(* CODESYS project system_dk.library
   Company: Beckhoff - DK
   DefaultNamespace: Tc3_System_DK
   Title: Tc3_System_DK
   Placeholder: Tc3_System_DK
   Author: HCP
   Version: 3.3.2.4

Project tree, tasks and I/O mapping:
  libraries: Tc2_EtherCAT, * (Beckhoff Automation GmbH); Tc2_IoFunctions, * (Beckhoff Automation GmbH); Tc2_Standard, * (Beckhoff Automation GmbH); Tc2_SUPS, * (Beckhoff Automation GmbH); Tc2_System, * (Beckhoff Automation GmbH); Tc2_Utilities, * (Beckhoff Automation GmbH); Tc3_Interfaces, * (Beckhoff Automation GmbH); Tc3_Module, * (Beckhoff Automation GmbH)
  DUTs/
  GVLs/
  POUs/
    BASE/
      FBs/
        [obsolete]/
          Basic/
            DUTs/
              data type ST_Basic
              data type ST_Basic_Status
            ITFs/
              interface I_Basic: M_nError, M_nReset, P_bAuto, P_bError, P_bManual, P_bReady, P_bReset, P_nErrorID
            function block FB_Basic [ST]: M_nError, M_nReset, P_bAuto, P_bError, P_bManual, P_bReady, P_bReset, P_nErrorID
        Base/
          DUTs/
            data type ST_Base
            data type ST_Base_Status
          ITFs/
            interface I_Base: M_nError, M_nReset, P_bError, P_bReady, P_bReset, P_nErrorID
          function block FB_Base [ST]: M_nError, M_nReset, P_bError, P_bReady, P_bReset, P_nErrorID
      GVLs/
        global variables GVL_Base
    SYSTEM/
      FBs/
        EtherCAT/
          DUTs/
            HW/
              data type ST_EtherCAT_HW_IN
              data type ST_EtherCAT_HW_TerminalDiagInfo
            data type ST_EtherCAT_DiagDk
            data type ST_EtherCAT_HW_Diag
          GVLs/
            global variables GVL_EtherCAT_Diag
          ITFs/
            interface I_EtherCAT_DiagDk: M_nCyclic, P_bEtherCAT_Ok, P_bWcError, P_nCfgSlaveCount, P_nDevState, P_nSlaveCounts
          function block FB_EtherCAT_DiagDk [ST]: M_nCyclic, M_sGetToken, P_bEtherCAT_Ok, P_bWcError, P_nCfgSlaveCount, P_nDevState, P_nSlaveCounts
        NovRam/
          DUTs/
            data type ST_NovRamDK
          ITFs/
            interface I_NovRamDK: M_nEnable
          function block FB_NovRamDK [ST]: M_nEnable, M_nRead, M_nWrite
        Persistent/
          DUTs/
            data type ST_WritePersistentDataDK
          ITFs/
            interface I_WritePersistentDataDK: M_n1_Second_UPS, M_nEnable, M_nWrite, P_bBusy, P_bPowerFailDetect, P_ePersistentMode, P_eSUPS_Mode, P_nWriteCNT
          function block FB_WritePersistentDataDK [ST]: M_n1_Second_UPS, M_nEnable, M_nWrite, P_bBusy, P_bPowerFailDetect, P_ePersistentMode, P_eSUPS_Mode, P_nWriteCNT
        System/
          DUTs/
            data type ST_SystemDK
          ITFs/
            interface I_SystemDK: M_nCerHost, M_nEnable, M_nGetTimeStampInMs, P_bIs_ARM, P_bIs_CE_Device, P_bIs_x64, P_bIs_x86, P_nAdsPort, P_nCycleTime, P_sHardwareSerialNumber, P_stDeviceIdentificationEx, P_sTwinCAT_Version
          function block FB_SystemDK [ST]: M_nCerHost, M_nEnable, M_nGetTimeStampInMs, P_bIs_ARM, P_bIs_CE_Device, P_bIs_x64, P_bIs_x86, P_nAdsPort, P_nCycleTime, P_sHardwareSerialNumber, P_stDeviceIdentificationEx, P_sTwinCAT_Version
  Version/
    global variables Global_Version
  VISUs/
*)

// POUs/BASE/FBs/[obsolete]/Basic/DUTs/ST_Basic
TYPE ST_Basic :
STRUCT
	bAuto: BOOL;
	bManual: BOOL;
	bReady: BOOL;
	bReset: BOOL;
	bError: BOOL;
	nErrorID: UDINT;
	nStatus: UDINT;	
	arr_nStatus: ARRAY[1..20] OF UDINT;
END_STRUCT
END_TYPE

// POUs/BASE/FBs/[obsolete]/Basic/DUTs/ST_Basic_Status
TYPE ST_Basic_Status :
STRUCT
	nError: UDINT;
	nReset:UDINT;
END_STRUCT
END_TYPE

// POUs/BASE/FBs/Base/DUTs/ST_Base
TYPE ST_Base :
STRUCT
	bReset: BOOL;
	bReady: BOOL;
	bError: BOOL;
	nErrorID: UDINT;
	arr_nStatus: ARRAY[1..20] OF UDINT;
END_STRUCT
END_TYPE

// POUs/BASE/FBs/Base/DUTs/ST_Base_Status
TYPE ST_Base_Status :
STRUCT
	nError: UDINT;
	nReset:UDINT;
END_STRUCT
END_TYPE

// POUs/SYSTEM/FBs/EtherCAT/DUTs/HW/ST_EtherCAT_HW_IN
TYPE ST_EtherCAT_HW_IN :
STRUCT
	AI_AmsNetId: AMSNETID;
	AI_nDevState: UINT;
	AI_nCfgSlaveCount: UINT;							
	AI_nSlaveCounts: UINT;								
	AI_nFrmXWcState: ARRAY[0..(GVL_EtherCAT_Diag.cMAX_NUMBERS_OF_EC_FRAMES -1)] OF UINT;
END_STRUCT
END_TYPE

// POUs/SYSTEM/FBs/EtherCAT/DUTs/HW/ST_EtherCAT_HW_TerminalDiagInfo
TYPE ST_EtherCAT_HW_TerminalDiagInfo :
STRUCT
	nAddr: UINT;
	sType: STRING(50);
	sName: STRING(50);
	nDeviceState: BYTE;
	nLinkState: BYTE;
	stTopologyDataEx: Tc2_EtherCAT.ST_TopologyDataEx;
END_STRUCT
END_TYPE

// POUs/SYSTEM/FBs/EtherCAT/DUTs/ST_EtherCAT_DiagDk
TYPE ST_EtherCAT_DiagDk EXTENDS ST_Basic:
STRUCT
	bEtherCAT_Ok: BOOL;				// ErtherCAT Ok signal
	bWcError: BOOL;
	nDevState: UINT;
	nCfgSlaveCount: UINT;							
	nSlaveCounts: UINT;								
END_STRUCT
END_TYPE

// POUs/SYSTEM/FBs/EtherCAT/DUTs/ST_EtherCAT_HW_Diag
TYPE ST_EtherCAT_HW_Diag :
STRUCT
	stAmsNetId: AMSNETID;			// EtherCAT Ams net id
	nState: WORD;					// EtherCAT master state
	sState: STRING;					// EtherCAT master state (string)
	nDevState: UINT;				// EtherCAT master DevState
	sDevState: STRING;				// EtherCAT master DevState (string)
	nCfgSlaveCount: UINT;			// Project configured slaves
	nSlaveCounts: UINT;				// Actual slave counts
	nMaxNumberOfSlaves: UINT;		// Max numbers of EtherCAT slaves
	bWcError: BOOL;					// Wc error
	bEtherCAT_Ok: BOOL;				// ErtherCAT Ok signal
	bReady: BOOL;					// Ready
	bError: BOOL;					// Error
	nErrorID: UDINT;				// Error ID
	arrFrmXWcState: ARRAY[0..(GVL_EtherCAT_Diag.cMAX_NUMBERS_OF_EC_FRAMES - 1)] OF UINT;		// EtherCAT master Wc state
	arrEcTerminalDiagInfo: ARRAY[1..GVL_EtherCAT_Diag.cMAX_NUMBERS_OF_EC_SLAVES] OF ST_EtherCAT_HW_TerminalDiagInfo;
END_STRUCT
END_TYPE

// POUs/SYSTEM/FBs/NovRam/DUTs/ST_NovRamDK
TYPE ST_NovRamDK EXTENDS ST_Basic :
STRUCT
	bEnable: BOOL;
END_STRUCT
END_TYPE

// POUs/SYSTEM/FBs/Persistent/DUTs/ST_WritePersistentDataDK
TYPE ST_WritePersistentDataDK EXTENDS ST_Basic :
STRUCT
	bWrite: BOOL;
	bBusy: BOOL;
	bPowerFailDetect: BOOL;
	nWriteCNT: UDINT;
END_STRUCT
END_TYPE

// POUs/SYSTEM/FBs/System/DUTs/ST_SystemDK
TYPE ST_SystemDK EXTENDS ST_Basic :
STRUCT
	bIs_CE_Device: BOOL;				// Is a CE Device
	bIs_ARM: BOOL;						// Is ARM runtime
	bIs_x86: BOOL;						// Is x86 runtime
	bIs_x64: BOOL;						// Is x64 runtime
	nAdsPort: UINT;						// Plc port nr
	nCycleTime: UDINT;					// Plc cycle time in 100nS
	bCerHost_Enable: BOOL;				// Enable CerHost
	bCerHost_Disable: BOOL;				// Disable CerHost
	sTwinCAT_Version: STRING(20);		// Runtime version
	sHardwareSerialNumber: STRING(20);	// Runtime hardware serial number
	stDeviceIdentificationEx: Tc2_Utilities.ST_DeviceIdentificationEx;		// Runtime info
END_STRUCT
END_TYPE

// POUs/BASE/GVLs/GVL_Base
VAR_GLOBAL CONSTANT
	cIDLE: UDINT:= 0;						//	0 = idle
	cCOUPLED: UDINT:= 1;					//	1 = coupled
	cSTARTING: UDINT:= 2;					//	2 = starting
	cRUNNING: UDINT:= 3;					//	3 = running
	cABORTED: UDINT:= 4;					//	4 = aborted
	cNO_HARDWARE_CONNECTED: UDINT:= 5;		// 	5 = no hardware connected

	cPOINTER_OR_INDEX_ERROR: UDINT:= 7;		//	7 = pointer or index error
	cMAPPING_ERROR: UDINT:= 8;				//	8 = mapping error
	cPARAMETER_ERROR: UDINT:= 9;			//	9 = parameter error
	cCOMPLETE: UDINT:= 10;					//	10 = complete
END_VAR

// POUs/SYSTEM/FBs/EtherCAT/GVLs/GVL_EtherCAT_Diag
{attribute 'qualified_only'}
VAR_GLOBAL CONSTANT
	cMAX_NUMBERS_OF_EC_SLAVES: UINT:= 1000;		// Max numbers of EtherCAT slaves
	cMAX_NUMBERS_OF_EC_FRAMES: UINT:= 10;		// Max numbers of EtherCAT frames
END_VAR

// Version/Global_Version
{attribute 'TcGenerated'}
{attribute 'no-analysis'}
{attribute 'linkalways'}
// This function has been automatically generated from the project information.
VAR_GLOBAL CONSTANT
	{attribute 'const_non_replaced'}
	stLibVersion_Tc3_System_DK : ST_LibVersion := (iMajor := 3, iMinor := 3, iBuild := 2, iRevision := 4, sVersion := '3.3.2.4');
END_VAR

// POUs/BASE/FBs/[obsolete]/Basic/ITFs/I_Basic
INTERFACE I_Basic

//	The result of the method is an unsigned double integer
//	0 = idle 
//	1 = coupled
//	2 = starting
//	3 = running
//	4 = aborted
// 	5 = no hardware connected
//  6 = Spare
//	7 = pointer or index error
//	8 = mapping error
//	9 = parameter error
//	10 = complete
//	Any other number = ErrorID
METHOD PUBLIC M_nError : UDINT
VAR_INPUT
	nErrorID: UDINT;
END_VAR
END_METHOD

//	The result of the method is an unsigned double integer
//	0 = idle 
//	1 = coupled
//	2 = starting
//	3 = running
//	4 = aborted
// 	5 = no hardware connected
//  6 = Spare
//	7 = pointer or index error
//	8 = mapping error
//	9 = parameter error
//	10 = complete
//	Any other number = ErrorID
METHOD PUBLIC M_nReset : UDINT
VAR_INPUT
	bExecute: BOOL;
END_VAR
END_METHOD

PROPERTY PUBLIC P_bAuto : BOOL
GET
END_GET
SET
END_SET
END_PROPERTY

PROPERTY PUBLIC P_bError : BOOL
GET
END_GET
END_PROPERTY

PROPERTY PUBLIC P_bManual : BOOL
GET
END_GET
SET
END_SET
END_PROPERTY

PROPERTY PUBLIC P_bReady : BOOL
GET
END_GET
SET
END_SET
END_PROPERTY

PROPERTY PUBLIC P_bReset : BOOL
GET
END_GET
END_PROPERTY

PROPERTY PUBLIC P_nErrorID : UDINT
GET
END_GET
END_PROPERTY

END_INTERFACE

// POUs/BASE/FBs/[obsolete]/Basic/FB_Basic
//------------------------------------------------------------------------------------------
//                                                                                        	
//***************************** Beckhoff TwinCAT Examples **********************************
//                                                                                        	
//************************************* WARNING ********************************************
// This program is only an example. If it is used as a control program in any real        	
// application, Beckhoff is not responsible for any malfunction, loss or damage           	
// which could arise by using this program!                                               	
//                                                                                        	
//*************************************  Program Info. *************************************
//                                                                                        	
// PLC program name:       	FB_Basic (FB)               	                           	
// Hardware platform:      	TwinCat v3.1.4012				                          	
// Modified by:            	Hans Chr. Pallesen 			                                  	
// Email:					h.pallesen@beckhoff.com	                                  	
//                                                                                        	
// ======================================================================================== 
//         Version       Date                        Remarks                              	
// ======================================================================================== 
//         1.0           17 feb 2013                 First release of this example        	
//         1.1           05 aug 2013                 Next release of this example        	
//         1.2           10 dec 2013                 Next release of this example        	
//         1.3           12 mar 2014                 Next release of this example        	
//         1.4           28 mar 2014                 Next release of this example        	
//         1.5           02 jun 2014                 Next release of this example        	
// ======================================================================================== 
//                                                                                        	
//******************************* Aims OF this PLC PROGRAM *********************************
//                                                                                        	
// Basic FB  						 			                               	
//																	                      	
//                                                                                        	
//----------------------------------------------------------------------------------------- 
FUNCTION_BLOCK FB_Basic IMPLEMENTS I_Basic
VAR
	_iIdx: INT;		// Temporary variabel - Index pointer
	
//*************************
// Property variables
//*************************
	_bReset: BOOL;
	_bAuto: BOOL := TRUE;
	_bManual: BOOL;
	_bError: BOOL;
	_nErrorID: UDINT;
	_bReady: BOOL;
	
//*************************
// Methods variable
//*************************
	_nResetState: UINT;
END_VAR

//	The result of the method is an unsigned double integer
//	0 = idle 
//	1 = coupled
//	2 = starting
//	3 = running
//	4 = aborted
// 	5 = no hardware connected
//  6 = Spare
//	7 = pointer or index error
//	8 = mapping error
//	9 = parameter error
//	10 = complete
//	Any other number = ErrorID
METHOD PUBLIC M_nError : UDINT
VAR_INPUT
	nErrorID: UDINT;
END_VAR
//**********************************
// Update error
//**********************************
IF _nResetState = 0 OR _nResetState = 4 THEN
	IF NOT _bError THEN
		_nErrorID:= nErrorID;
		_bError:= TRUE;
	END_IF
END_IF

M_nError:= cCOMPLETE;
END_METHOD

//	The result of the method is an unsigned double integer
//	0 = idle 
//	1 = coupled
//	2 = starting
//	3 = running
//	4 = aborted
// 	5 = no hardware connected
//  6 = Spare
//	7 = pointer or index error
//	8 = mapping error
//	9 = parameter error
//	10 = complete
//	Any other number = ErrorID
METHOD PUBLIC M_nReset : UDINT
VAR_INPUT
	bExecute: BOOL;
END_VAR
// Reset handling
CASE _nResetState OF

	000:	// Wait for execute
			M_nReset:= cIDLE;
			IF bExecute THEN
				_bReset:= TRUE;
				_nResetState:= _nResetState +1;
			ELSE
				_bReset:= FALSE;
			END_IF

	001:	// Reset update
			M_nReset:= cRUNNING;
			_nResetState:= _nResetState +1;
		
	002:	// Reset error flag
			M_nReset:= cRUNNING;
			_bError:= FALSE;
			_nErrorID:= 16#00;
			_nResetState:= _nResetState +1;
	
	003:	// Reset update
			M_nReset:= cRUNNING;
			_nResetState:= _nResetState +1;
		
	004:	// Wait for not execute
			IF bExecute THEN
				M_nReset:= cCOMPLETE;
			ELSE
				M_nReset:= cCOMPLETE;
				_bReset:= FALSE;
				_nResetState:= 000;
			END_IF

ELSE
		_nResetState:= 000;
END_CASE
END_METHOD

PROPERTY PUBLIC P_bAuto : BOOL
GET
P_bAuto:= _bAuto;
END_GET
SET
_bAuto:= P_bAuto;
END_SET
END_PROPERTY

PROPERTY PUBLIC P_bError : BOOL
GET
P_bError:= _bError;
END_GET
END_PROPERTY

PROPERTY PUBLIC P_bManual : BOOL
GET
P_bManual:= _bManual;
END_GET
SET
_bManual:= P_bManual;
END_SET
END_PROPERTY

PROPERTY PUBLIC P_bReady : BOOL
GET
P_bReady:= _bReady;
END_GET
SET
PUBLIC 
VAR
END_VAR
_bReady:= P_bReady;
END_SET
END_PROPERTY

PROPERTY PUBLIC P_bReset : BOOL
GET
P_bReset:= _bReset;
END_GET
END_PROPERTY

PROPERTY PUBLIC P_nErrorID : UDINT
GET
P_nErrorID:= _nErrorID;
END_GET
END_PROPERTY

END_FUNCTION_BLOCK

// POUs/BASE/FBs/Base/ITFs/I_Base
INTERFACE I_Base

//	The result of the method is an unsigned double integer
//	0 = idle 
//	1 = coupled
//	2 = starting
//	3 = running
//	4 = aborted
// 	5 = no hardware connected
//  6 = Spare
//	7 = pointer or index error
//	8 = mapping error
//	9 = parameter error
//	10 = complete
//	Any other number = ErrorID
METHOD PUBLIC M_nError : UDINT
VAR_INPUT
	nErrorID: UDINT;
END_VAR
END_METHOD

//	The result of the method is an unsigned double integer
//	0 = idle 
//	1 = coupled
//	2 = starting
//	3 = running
//	4 = aborted
// 	5 = no hardware connected
//  6 = Spare
//	7 = pointer or index error
//	8 = mapping error
//	9 = parameter error
//	10 = complete
//	Any other number = ErrorID
METHOD PUBLIC M_nReset : UDINT
VAR_INPUT
	bExecute: BOOL;
END_VAR
END_METHOD

PROPERTY PUBLIC P_bError : BOOL
GET
END_GET
END_PROPERTY

PROPERTY PUBLIC P_bReady : BOOL
GET
END_GET
SET
END_SET
END_PROPERTY

PROPERTY PUBLIC P_bReset : BOOL
GET
END_GET
END_PROPERTY

PROPERTY PUBLIC P_nErrorID : UDINT
GET
END_GET
END_PROPERTY

END_INTERFACE

// POUs/BASE/FBs/Base/FB_Base
//------------------------------------------------------------------------------------------
//                                                                                        	
//***************************** Beckhoff TwinCAT Examples **********************************
//                                                                                        	
//************************************* WARNING ********************************************
// This program is only an example. If it is used as a control program in any real        	
// application, Beckhoff is not responsible for any malfunction, loss or damage           	
// which could arise by using this program!                                               	
//                                                                                        	
//*************************************  Program Info. *************************************
//                                                                                        	
// PLC program name:       	FB_Basic (FB)               	                           	
// Hardware platform:      	TwinCat v3.1.4020				                          	
// Modified by:            	Hans Chr. Pallesen 			                                  	
// Email:					h.pallesen@beckhoff.com	                                  	
//                                                                                        	
// ======================================================================================== 
//         Version       Date                        Remarks                              	
// ======================================================================================== 
//         1.0           02 mar 2019                 First release of this example        	
// ======================================================================================== 
//                                                                                        	
//******************************* Aims OF this PLC PROGRAM *********************************
//                                                                                        	
// Base FB  						 			                               	
//																	                      	
//                                                                                        	
//----------------------------------------------------------------------------------------- 
FUNCTION_BLOCK FB_Base IMPLEMENTS I_Base
VAR
	
//*************************
// Property variables
//*************************
	_bReset: BOOL;
	_bError: BOOL;
	_nErrorID: UDINT;
	_bReady: BOOL;

//*************************
// Methodes variables
//*************************
	_nResetState: UINT;
	
END_VAR

//	The result of the method is an unsigned double integer
//	0 = idle 
//	1 = coupled
//	2 = starting
//	3 = running
//	4 = aborted
// 	5 = no hardware connected
//  6 = Spare
//	7 = pointer or index error
//	8 = mapping error
//	9 = parameter error
//	10 = complete
//	Any other number = ErrorID
METHOD PUBLIC M_nError : UDINT
VAR_INPUT
	nErrorID: UDINT;
END_VAR
//**********************************
// Update error
//**********************************
IF _nResetState = 0 OR _nResetState = 4 THEN
	IF NOT _bError THEN
		_nErrorID:= nErrorID;
		_bError:= TRUE;
	END_IF
END_IF

M_nError:= cCOMPLETE;
END_METHOD

//	The result of the method is an unsigned double integer
//	0 = idle 
//	1 = coupled
//	2 = starting
//	3 = running
//	4 = aborted
// 	5 = no hardware connected
//  6 = Spare
//	7 = pointer or index error
//	8 = mapping error
//	9 = parameter error
//	10 = complete
//	Any other number = ErrorID
METHOD PUBLIC M_nReset : UDINT
VAR_INPUT
	bExecute: BOOL;
END_VAR
VAR_INST
	_FB_Base_M_nReset_nState: UINT;
END_VAR
// Reset handling
CASE _FB_Base_M_nReset_nState OF

	000:	// Wait for execute
			M_nReset:= cIDLE;
			IF bExecute THEN
				_bReset:= TRUE;
				_FB_Base_M_nReset_nState:= _FB_Base_M_nReset_nState +1;
			ELSE
				_bReset:= FALSE;
			END_IF

	001:	// Reset update
			M_nReset:= cRUNNING;
			_FB_Base_M_nReset_nState:= _FB_Base_M_nReset_nState +1;
		
	002:	// Reset error flag
			M_nReset:= cRUNNING;
			_bError:= FALSE;
			_nErrorID:= 16#00;
			_FB_Base_M_nReset_nState:= _FB_Base_M_nReset_nState +1;
	
	003:	// Reset update
			M_nReset:= cRUNNING;
			_FB_Base_M_nReset_nState:= _FB_Base_M_nReset_nState +1;
		
	004:	// Wait for not execute
			IF bExecute THEN
				M_nReset:= cCOMPLETE;
			ELSE
				M_nReset:= cCOMPLETE;
				_bReset:= FALSE;
				_FB_Base_M_nReset_nState:= 000;
			END_IF

ELSE
		_FB_Base_M_nReset_nState:= 000;
END_CASE
END_METHOD

{attribute 'monitoring' := 'variable'}
PROPERTY PUBLIC P_bError : BOOL
GET
P_bError:= _bError;
END_GET
END_PROPERTY

{attribute 'monitoring' := 'variable'}
PROPERTY PUBLIC P_bReady : BOOL
GET
P_bReady:= _bReady;
END_GET
SET
PUBLIC 
VAR
END_VAR
_bReady:= P_bReady;
END_SET
END_PROPERTY

{attribute 'monitoring' := 'variable'}
PROPERTY PUBLIC P_bReset : BOOL
GET
P_bReset:= _bReset;
END_GET
END_PROPERTY

{attribute 'monitoring' := 'variable'}
PROPERTY PUBLIC P_nErrorID : UDINT
GET
P_nErrorID:= _nErrorID;
END_GET
END_PROPERTY

END_FUNCTION_BLOCK

// POUs/SYSTEM/FBs/EtherCAT/ITFs/I_EtherCAT_DiagDk
INTERFACE I_EtherCAT_DiagDk EXTENDS I_Basic

//	The result of the method is an unsigned double integer
//	0 = idle 
//	1 = coupled
//	2 = starting
//	3 = running
//	4 = aborted
// 	5 = no hardware connected
//  6 = Spare
//	7 = pointer or index error
//	8 = mapping error
//	9 = parameter error
//	10 = complete
//	Any other number = ErrorID
METHOD PUBLIC M_nCyclic : UDINT
VAR_INPUT
	bEnable: BOOL;
	pEtherCAT_Diag: POINTER TO ST_EtherCAT_HW_Diag;	
END_VAR
END_METHOD

PROPERTY PUBLIC P_bEtherCAT_Ok : BOOL
GET
END_GET
SET
END_SET
END_PROPERTY

PROPERTY PUBLIC P_bWcError : bool
GET
END_GET
END_PROPERTY

PROPERTY PUBLIC P_nCfgSlaveCount : UINT
GET
END_GET
END_PROPERTY

PROPERTY PUBLIC P_nDevState : UINT
GET
END_GET
END_PROPERTY

PROPERTY PUBLIC P_nSlaveCounts : UINT
GET
END_GET
END_PROPERTY

END_INTERFACE

// POUs/SYSTEM/FBs/EtherCAT/FB_EtherCAT_DiagDk
//------------------------------------------------------------------------------------------
//                                                                                        	
//***************************** Beckhoff TwinCAT Examples **********************************
//                                                                                        	
//************************************* WARNING ********************************************
// This program is only an example. If it is used as a control program in any real        	
// application, Beckhoff is not responsible for any malfunction, loss or damage           	
// which could arise by using this program!                                               	
//                                                                                        	
//*************************************  Program Info. *************************************
//                                                                                        	
// PLC program name:       	FB_EtherCAT_Diag (FB)                                          	
// Hardware platform:      	TwinCAT v3.1.4022				                          	
// Modified by:            	Hans Chr. Pallesen 			                                  	
// Email:					h.pallesen@beckhoff.com	                                  	
//                                                                                        	
// ======================================================================================== 
//         Version       Date                        Remarks                              	
// ======================================================================================== 
//         1.0           12 dec 2016                 First release of this example        	
// ======================================================================================== 
//                                                                                        	
//******************************* Aims OF this PLC PROGRAM *********************************
//                                                                                        	
// EtherCAT diagnose				 			                                      	
//																	                      	
//                                                                                        	
//----------------------------------------------------------------------------------------- 
FUNCTION_BLOCK FB_EtherCAT_DiagDk EXTENDS FB_Basic IMPLEMENTS I_EtherCAT_DiagDk
VAR
	bFirstScan: BOOL:= TRUE;
	stIN AT %I*: ST_EtherCAT_HW_IN;
	
	_pEtherCAT_Diag: POINTER TO ST_EtherCAT_HW_Diag;	
	_bWcError: BOOL;
	_nDeviceNumber: UINT:= 1;
	_nSlaves: UINT;
	
	arrEcSlaveConfigData: ARRAY[1..GVL_EtherCAT_Diag.cMAX_NUMBERS_OF_EC_SLAVES] OF Tc2_EtherCAT.ST_EcSlaveConfigData;
	arrEcSlaveState: ARRAY[1..GVL_EtherCAT_Diag.cMAX_NUMBERS_OF_EC_SLAVES] OF Tc2_EtherCAT.ST_EcSlaveState;
	arrTopologyDataEx: ARRAY[1..GVL_EtherCAT_Diag.cMAX_NUMBERS_OF_EC_SLAVES] OF Tc2_EtherCAT.ST_TopologyDataEx;
	arrEcSlaveName: ARRAY[1..GVL_EtherCAT_Diag.cMAX_NUMBERS_OF_EC_SLAVES] OF STRING;;
	arrFrmXWcStateOld: ARRAY[0..(GVL_EtherCAT_Diag.cMAX_NUMBERS_OF_EC_FRAMES -1)] OF UINT;
	arrFrmXWcStateInit: ARRAY[0..(GVL_EtherCAT_Diag.cMAX_NUMBERS_OF_EC_FRAMES -1)] OF UINT;
	
	fbEcGetMasterState: Tc2_EtherCAT.FB_EcGetMasterState;
	fbEcGetConfSlaves: Tc2_EtherCAT.FB_EcGetConfSlaves;
	fbEcGetAllSlaveStates: Tc2_EtherCAT.FB_EcGetAllSlaveStates;
	fbEcGetSlaveIdentity: Tc2_EtherCAT.FB_EcGetSlaveIdentity;
	fbEcGetSlaveTopologyInfo: Tc2_EtherCAT.FB_EcGetSlaveTopologyInfo;
END_VAR

//	The result of the method is an unsigned double integer
//	0 = idle 
//	1 = coupled
//	2 = starting
//	3 = running
//	4 = aborted
// 	5 = no hardware connected
//  6 = Spare
//	7 = pointer or index error
//	8 = mapping error
//	9 = parameter error
//	10 = complete
//	Any other number = ErrorID
METHOD PUBLIC M_nCyclic : UDINT
VAR_INPUT
	bEnable: BOOL;
	pEtherCAT_Diag: POINTER TO ST_EtherCAT_HW_Diag;	
END_VAR
VAR_INST
	i: UINT;
	iState: INT;
	sString: STRING;
	nCNT: INT;
	nDevStateOld: UINT;
	nSlaveCountsOld: UINT;								
	fbEnable_R_TRIG: Tc2_Standard.R_TRIG;
	fbDelay_TON: Tc2_Standard.TON;
	fbReadyDelay_TON: Tc2_Standard.TON;
END_VAR
// Local variable
_pEtherCAT_Diag:= pEtherCAT_Diag;

// Reset
IF _bReset THEN
	IF P_bError THEN
		iState:= 000;
	END_IF	
END_IF

// Pointer check
IF _pEtherCAT_Diag = 16#00 THEN
	_bReady:= FALSE;
	iState:= 000;
	M_nCyclic:= cPOINTER_OR_INDEX_ERROR;
	RETURN;
END_IF

// Update EtherCAT State
pEtherCAT_Diag^.nState:= fbEcGetMasterState.state;	
pEtherCAT_Diag^.sState := F_ConvStateToString(fbEcGetMasterState.state);
pEtherCAT_Diag^.nDevState:= stIN.AI_nDevState; 
pEtherCAT_Diag^.sDevState:= F_ConvMasterDevStateToString(stIN.AI_nDevState);
pEtherCAT_Diag^.nSlaveCounts:= stIN.AI_nSlaveCounts;
pEtherCAT_Diag^.nCfgSlaveCount:= stIN.AI_nCfgSlaveCount;

// EtherCAT Mapping check
IF stIN.AI_AmsNetId[0] = 0 AND stIN.AI_AmsNetId[5] = 0 THEN
	_bReady:= FALSE;
	iState:= 000;
	M_nCyclic:= cMAPPING_ERROR;
	RETURN;
END_IF

// Mapping check
IF stIN.AI_nSlaveCounts = 0 OR stIN.AI_nCfgSlaveCount = 0 THEN
	_bReady:= FALSE;
	iState:= 000;
	M_nCyclic:= cMAPPING_ERROR;
	RETURN;
END_IF

// Not Enable
fbEnable_R_TRIG(CLK:= NOT bEnable, Q=> );
IF fbEnable_R_TRIG.Q THEN
	_bReady:= FALSE;
	iState:= 000;
	RETURN;
END_IF

// Update GVL data
pEtherCAT_Diag^.stAmsNetId:= stIN.AI_AmsNetId;
pEtherCAT_Diag^.bReady:= P_bReady;
pEtherCAT_Diag^.bError:= P_bError;
pEtherCAT_Diag^.nErrorID:= P_nErrorID;
pEtherCAT_Diag^.nMaxNumberOfSlaves:= GVL_EtherCAT_Diag.cMAX_NUMBERS_OF_EC_SLAVES;
pEtherCAT_Diag^.arrFrmXWcState:= stIN.AI_nFrmXWcState;


// State maschine
CASE iState OF
	
	000:	// Init
			M_nCyclic:= cSTARTING;
			fbEcGetMasterState(bExecute:= FALSE); 
			fbEcGetConfSlaves(pArrEcConfSlaveInfo:= ADR(arrEcSlaveConfigData), cbBufLen:= SIZEOF(arrEcSlaveConfigData), bExecute:= FALSE); 
			fbEcGetAllSlaveStates(pStateBuf:= ADR(arrEcSlaveState), cbBufLen:= SIZEOF(arrEcSlaveState), bExecute:= FALSE); 
			fbEcGetSlaveTopologyInfo(pAddrBuf:= ADR(arrTopologyDataEx), cbBufLen:= SIZEOF(arrTopologyDataEx), bExecute:= FALSE); 
			fbEcGetSlaveIdentity(bExecute:= FALSE);
			fbDelay_TON(IN:= FALSE, PT:= , Q=> , ET=> );
			fbReadyDelay_TON(IN:= FALSE, PT:= , Q=> , ET=> );
			P_bReady:= FALSE;
			iState:= iState +1;	

	001:	// Wait for enable + delay	
			M_nCyclic:= cIDLE;
			fbDelay_TON(IN:= bEnable, PT:= T#200MS, Q=> , ET=> );
			IF fbDelay_TON.Q THEN
				IF bFirstScan THEN
					iState:= iState +1;
				ELSE
					iState:= iState +2;
				END_IF	
			END_IF
		
	002:	// Get Conf Slaves
			M_nCyclic:= cRUNNING;
			fbEcGetConfSlaves(
				sNetId:= F_CreateAmsNetId(stIN.AI_AmsNetId), 
				pArrEcConfSlaveInfo:= ADR(arrEcSlaveConfigData), 
				cbBufLen:= SIZEOF(arrEcSlaveConfigData), 
				bExecute:= TRUE, 
				tTimeout:= , 
				bBusy=> , 
				bError=> , 
				nErrorId=> , 
				nSlaves=> );
				
			// Error	
			IF fbEcGetConfSlaves.bError THEN
				M_nError(nErrorID:= fbEcGetConfSlaves.nErrorId);
				M_nCyclic:= fbEcGetConfSlaves.nErrorId;
			ELSE
				// Done
				IF NOT fbEcGetConfSlaves.bBusy THEN
					fbEcGetConfSlaves(pArrEcConfSlaveInfo:= ADR(arrEcSlaveConfigData), cbBufLen:= SIZEOF(arrEcSlaveConfigData), bExecute:= FALSE);
					iState:= iState +1;	
				END_IF
			END_IF

	003:	// Get Master state
			M_nCyclic:= cRUNNING;
			fbEcGetMasterState(
				sNetId:= F_CreateAmsNetId(stIN.AI_AmsNetId), 
				bExecute:= TRUE, 
				tTimeout:= , 
				bBusy=> , 
				bError=> , 
				nErrId=> , 
				state=> );

			// Error
			IF fbEcGetMasterState.bError THEN
				M_nError(nErrorID:= fbEcGetMasterState.nErrId);
				M_nCyclic:= fbEcGetMasterState.nErrId;
			ELSE
				// Done
				IF NOT fbEcGetMasterState.bBusy THEN
					fbEcGetMasterState(bExecute:= FALSE); 
					iState:= iState +1;	
				END_IF
			END_IF

	004:	// Get all slave states
			M_nCyclic:= cRUNNING;
			fbEcGetAllSlaveStates(
				sNetId:= F_CreateAmsNetId(stIN.AI_AmsNetId),
				pStateBuf:= ADR(arrEcSlaveState), 
				cbBufLen:= SIZEOF(arrEcSlaveState), 
				bExecute:= TRUE, 
				tTimeout:= , 
				bBusy=> , 
				bError=> , 
				nErrId=> , 
				nSlaves=>);
	
			// Error
			IF fbEcGetAllSlaveStates.bError THEN
				M_nError(nErrorID:= fbEcGetAllSlaveStates.nErrId);
				M_nCyclic:= fbEcGetAllSlaveStates.nErrId;
			ELSE
				// Done	
				IF NOT fbEcGetAllSlaveStates.bBusy THEN
					_nSlaves:= fbEcGetAllSlaveStates.nSlaves;
					IF _nSlaves > GVL_EtherCAT_Diag.cMAX_NUMBERS_OF_EC_SLAVES THEN
						_nSlaves:= GVL_EtherCAT_Diag.cMAX_NUMBERS_OF_EC_SLAVES;
					END_IF
					fbEcGetAllSlaveStates(pStateBuf:= ADR(arrEcSlaveState), cbBufLen:= SIZEOF(arrEcSlaveState), bExecute:= FALSE);
					iState:= iState +1;	
				END_IF 
			END_IF		
				
	005:	// Get device name	
			M_nCyclic:= cRUNNING;
			IF _nDeviceNumber <= _nSlaves THEN
				fbEcGetSlaveIdentity(
					sNetId:= F_CreateAmsNetId(stIN.AI_AmsNetId), 
					nSlaveAddr:= arrEcSlaveConfigData[_nDeviceNumber].nAddr, 
					bExecute:= TRUE, 
					tTimeout:= , 
					bBusy=> , 
					bError=> , 
					nErrId=> , 
					identity=> );
		
					// Error
					IF fbEcGetSlaveIdentity.bError THEN
						M_nError(nErrorID:= fbEcGetSlaveIdentity.nErrId);
						M_nCyclic:= fbEcGetSlaveIdentity.nErrId;
					ELSE
						// Done	
						IF NOT fbEcGetSlaveIdentity.bBusy THEN
							arrEcSlaveName[_nDeviceNumber]:= F_ConvProductCodeToString(fbEcGetSlaveIdentity.identity);	
							fbEcGetSlaveIdentity(bExecute:= FALSE); 
							_nDeviceNumber:= _nDeviceNumber +1;
							iState:= iState +1;	
						END_IF 
					END_IF		
				
			ELSE
				iState:= iState +2;	
			END_IF

	006:	// Next device
			M_nCyclic:= cRUNNING;
			iState:= iState -1;	
	
	007:	// Update status
			M_nCyclic:= cRUNNING;
			
			// Slave counts Wc state update
			FOR i:= 1 TO GVL_EtherCAT_Diag.cMAX_NUMBERS_OF_EC_FRAMES DO
				pEtherCAT_Diag^.arrFrmXWcState[i]:= stIN.AI_nFrmXWcState[i];
			END_FOR
			
			// Slave counts status update
			FOR i:= 1 TO _nSlaves DO
				pEtherCAT_Diag^.arrEcTerminalDiagInfo[i].nAddr:= arrEcSlaveConfigData[i].nAddr;
				pEtherCAT_Diag^.arrEcTerminalDiagInfo[i].sType:= arrEcSlaveName[i];
				
				// Read string until '('
				sString:= M_sGetToken(pSrcAddr:= ADR(arrEcSlaveConfigData[i].sName), sDelim:= '(', nToken:= 1); 
				IF sString = '' THEN
					pEtherCAT_Diag^.arrEcTerminalDiagInfo[i].sName:= arrEcSlaveConfigData[i].sName;
				ELSE
					sString:= Tc2_Standard.CONCAT(sString,'(');
					sString:= Tc2_Standard.CONCAT(sString,Tc2_Standard.MID(_pEtherCAT_Diag^.arrEcTerminalDiagInfo[i].sType, 6, 1));
					sString:= Tc2_Standard.CONCAT(sString,')');
					pEtherCAT_Diag^.arrEcTerminalDiagInfo[i].sName:= sString;
				END_IF
				pEtherCAT_Diag^.arrEcTerminalDiagInfo[i].nDeviceState:= arrEcSlaveState[i].deviceState;
				pEtherCAT_Diag^.arrEcTerminalDiagInfo[i].nLinkState:= arrEcSlaveState[i].linkState;
				
			END_FOR
			bFirstScan:= FALSE; 
			iState:= iState +1;	
			
	008:	// Update devece state once more			
			M_nCyclic:= cRUNNING;
			nCNT:= nCNT +1;
			IF nCNT >= 2 THEN
				nCNT:= 0;
				iState:= iState +1;	
			ELSE
				iState:= 000;	
			END_IF
			
	009:	// Read slave TopologyDataEx		
			M_nCyclic:= cRUNNING;
			fbEcGetSlaveTopologyInfo(
				sNetId:= F_CreateAmsNetId(stIN.AI_AmsNetId), 
				pAddrBuf:= ADR(arrTopologyDataEx), 
				cbBufLen:= SIZEOF(arrTopologyDataEx), 
				bExecute:= TRUE, 
				tTimeout:= , 
				bBusy=> , 
				bError=> , 
				nErrId=> , 
				nSlaves=> );
	
			// Error
			IF fbEcGetSlaveTopologyInfo.bError THEN
				M_nError(nErrorID:= fbEcGetSlaveTopologyInfo.nErrId);
				M_nCyclic:= fbEcGetSlaveTopologyInfo.nErrId;
			ELSE
				// Done	
				IF NOT fbEcGetSlaveTopologyInfo.bBusy THEN
					fbEcGetSlaveTopologyInfo(pAddrBuf:= ADR(arrTopologyDataEx), cbBufLen:= SIZEOF(arrTopologyDataEx), bExecute:= FALSE); 
					FOR i:= 1 TO _nSlaves DO
						pEtherCAT_Diag^.arrEcTerminalDiagInfo[i].stTopologyDataEx:= arrTopologyDataEx[i];	
					END_FOR
					iState:= iState +1;	
				END_IF 
			END_IF		

	010:	// Update EtherCAT state
			M_nCyclic:= cRUNNING;
			fbReadyDelay_TON(IN:= TRUE, PT:= T#200MS, Q=> , ET=> );
	
			// Wait for Slave counts change
			IF nSlaveCountsOld <> stIN.AI_nSlaveCounts THEN
				nSlaveCountsOld:= stIN.AI_nSlaveCounts;
				iState:= 000;
				RETURN;
			ELSE	
				// Wait for DevState change
				IF nDevStateOld <> stIN.AI_nDevState THEN
					nDevStateOld:= stIN.AI_nDevState;
					iState:= 000;
					RETURN;
				ELSE
					// Wait for Wc state change			
					IF MEMCMP(pBuf1:= ADR(arrFrmXWcStateOld), pBuf2:= ADR(pEtherCAT_Diag^.arrFrmXWcState), n:= SIZEOF(arrFrmXWcStateOld)) <> 0 THEN
						Tc2_System.MEMCPY(destAddr:= ADR(arrFrmXWcStateOld), srcAddr:= ADR(pEtherCAT_Diag^.arrFrmXWcState), n:= SIZEOF(arrFrmXWcStateOld));
						iState:= 000;
						RETURN;
					END_IF
				END_IF	
			END_IF

			// Error
			IF P_bError THEN
				P_bReady:= FALSE;
				M_nCyclic:= P_nErrorID;
			ELSE	
				IF fbReadyDelay_TON.Q THEN
					P_bReady:= TRUE;
				END_IF	
				M_nCyclic:= cCOMPLETE;
			END_IF

ELSE
	iState:= 000;
END_CASE

// Update Wc error
IF MEMCMP(pBuf1:= ADR(_pEtherCAT_Diag^.arrFrmXWcState), pBuf2:= ADR(arrFrmXWcStateInit), n:= SIZEOF(_pEtherCAT_Diag^.arrFrmXWcState)) = 0 THEN
	_pEtherCAT_Diag^.bWcError:= FALSE;
	_bWcError:= FALSE;
ELSE
	_pEtherCAT_Diag^.bWcError:= TRUE;
	_bWcError:= TRUE;
END_IF
END_METHOD

//------------------------------------------------------------------------------------------
//                                                                                        	
//***************************** Beckhoff TwinCAT Examples **********************************
//                                                                                        	
//************************************* WARNING ********************************************
// This program is only an example. If it is used as a control program in any real        	
// application, Beckhoff is not responsible for any malfunction, loss or damage           	
// which could arise by using this program!                                               	
//                                                                                        	
//*************************************  Program Info. *************************************
//                                                                                        	
// PLC program name:       F_sGetToken (FUN)               	                           	
// Hardware platform:      TwinCAT v3.1.4018.26				                          	
// Modified by:            Hans Chr. Pallesen 			                                  	
//                                                                                        	
// ======================================================================================== 
//         Version       Date                        Remarks                              	
// ======================================================================================== 
//         1.00          14 feb 2016                 First release of this example        	
// ======================================================================================== 
//                                                                                        	
//******************************* Aims OF this PLC PROGRAM *********************************
//                                                                                        	
// 	Description:																
//																			
//    sAllTokens         		iToken   	sDelim  	Returns     Notes						
//   "William M Rawls"    	   1      		   " "    	"William" 	First word				
//   "William M Rawls"    	   2      		   " "     	"M"         Second word					
//   "William M Rawls"     	   3      		   " "     	"Rawls"     Third word				
//   "William M Rawls"    	   4      		   " "     	""          No forth word					
//   "William M Rawls"    	   0      		   " "     	""          Zeroth token is always empty		
//   "William M Rawls"   	   -1      	 	   " "     	""          Negative tokesn always empty		
//   "William M Rawls"    	   1      		   ""      	""          No delimiter ? Token empty		
//----------------------------------------------------------------------------------------- 
METHOD PRIVATE M_sGetToken: Tc2_System.T_MaxString
VAR_INPUT
	pSrcAddr: POINTER TO Tc2_System.T_MaxString;
  	sDelim: STRING;
	nToken: UINT;
END_VAR
VAR
// Temporary Variables 
	nCurTokenLocation: INT;
END_VAR
IF nToken < 1 OR Tc2_Standard.LEN(sDelim) < 1 THEN
	// Negative OR zeroth token OR empty delimiter strings mean an empty token 
	M_sGetToken:= '';
 	RETURN;
ELSE
	IF nToken = 1 THEN
	// Quickly extract the first token 
	nCurTokenLocation:= Tc2_Standard.FIND(pSrcAddr^, sDelim);
	   	IF nCurTokenLocation > 1 THEN
	   		M_sGetToken:= Tc2_Standard.LEFT(pSrcAddr^, nCurTokenLocation - 1);
	   	ELSE
			M_sGetToken:= pSrcAddr^;
	    END_IF
	ELSE
		// FIND the Nth token 
		REPEAT
			nCurTokenLocation:= Tc2_Standard.FIND(pSrcAddr^, sDelim);
			IF nCurTokenLocation = 0 THEN
				M_sGetToken:= '';
				RETURN;
			ELSE
				pSrcAddr:= pSrcAddr + INT_TO_DWORD(nCurTokenLocation -1) + INT_TO_DWORD(Tc2_Standard.LEN(sDelim));
			END_IF
	
			nToken:= nToken - 1;
			UNTIL nToken = 1
		END_REPEAT;

		// Extract the Nth token (Which is the next token AT this point) 
		nCurTokenLocation:= Tc2_Standard.FIND(pSrcAddr^, sDelim);
		IF nCurTokenLocation > 0 THEN
			M_sGetToken:= Tc2_Standard.LEFT(pSrcAddr^, nCurTokenLocation - 1);
			RETURN;
		ELSE
			M_sGetToken:= pSrcAddr^;
		   	RETURN;
		END_IF
	END_IF
END_IF
END_METHOD

{attribute 'monitoring' := 'variable'}
PROPERTY PUBLIC P_bEtherCAT_Ok : BOOL
GET
// Pointer check
IF _pEtherCAT_Diag <> 16#00 THEN
	P_bEtherCAT_Ok:= _pEtherCAT_Diag^.bEtherCAT_Ok;
ELSE
	P_bEtherCAT_Ok:= FALSE;
END_IF
END_GET
SET
PUBLIC 
VAR
END_VAR
// Pointer check
IF _pEtherCAT_Diag <> 16#00 THEN
	_pEtherCAT_Diag^.bEtherCAT_Ok:= P_bEtherCAT_Ok;
END_IF
END_SET
END_PROPERTY

{attribute 'monitoring' := 'variable'}
PROPERTY PUBLIC P_bWcError : bool
GET
P_bWcError:= _bWcError;
END_GET
END_PROPERTY

{attribute 'monitoring' := 'variable'}
PROPERTY PUBLIC P_nCfgSlaveCount : UINT
GET
// Pointer check
IF _pEtherCAT_Diag <> 16#00 THEN
	P_nCfgSlaveCount:= _pEtherCAT_Diag^.nCfgSlaveCount;
END_IF
END_GET
END_PROPERTY

{attribute 'monitoring' := 'variable'}
PROPERTY PUBLIC P_nDevState : UINT
GET
// Pointer check
IF _pEtherCAT_Diag <> 16#00 THEN
	P_nDevState:= _pEtherCAT_Diag^.nDevState;
END_IF
END_GET
END_PROPERTY

{attribute 'monitoring' := 'variable'}
PROPERTY PUBLIC P_nSlaveCounts : UINT
GET
// Pointer check
IF _pEtherCAT_Diag <> 16#00 THEN
	P_nSlaveCounts:= _pEtherCAT_Diag^.nSlaveCounts;
END_IF
END_GET
END_PROPERTY

END_FUNCTION_BLOCK

// POUs/SYSTEM/FBs/NovRam/ITFs/I_NovRamDK
INTERFACE I_NovRamDK EXTENDS I_Basic

//	The result of the method is an unsigned double integer
//	0 = idle 
//	1 = coupled
//	2 = starting
//	3 = running
//	4 = aborted
// 	5 = no hardware connected
//  6 = Spare
//	7 = pointer or index error
//	8 = mapping error
//	9 = parameter error
//	10 = complete
//	Any other number = ErrorID
METHOD M_nEnable : UDINT
VAR_INPUT
	bExecute: BOOL;
	nDevId: UINT;
	nMB_Offset: UINT;
	nMB_Size: UINT;
END_VAR
END_METHOD

END_INTERFACE

// POUs/SYSTEM/FBs/NovRam/FB_NovRamDK
//------------------------------------------------------------------------------------------
//                                                                                        	
//***************************** Beckhoff TwinCAT Examples **********************************
//                                                                                        	
//************************************* WARNING ********************************************
// This program is only an example. If it is used as a control program in any real        	
// application, Beckhoff is not responsible for any malfunction, loss or damage           	
// which could arise by using this program!                                               	
//                                                                                        	
//*************************************  Program Info. *************************************
//                                                                                        	
// PLC program name:       	FB_NovRamDK (FB)               	                           	
// Hardware platform:      	TwinCat v3.1.4022				                          	
// Modified by:            	Hans Chr. Pallesen 			                                  	
// Email:					h.pallesen@beckhoff.com	                                  	
//                                                                                        	
// ======================================================================================== 
//         Version       Date                        Remarks                              	
// ======================================================================================== 
//         1.0           27 nov 2013                 First release of this example        	
// ======================================================================================== 
//                                                                                        	
//******************************* Aims OF this PLC PROGRAM *********************************
//                                                                                        	
//	Read/Write to NovRam																	                      	
//                                                                                        	
//----------------------------------------------------------------------------------------- 
FUNCTION_BLOCK FB_NovRamDK EXTENDS FB_Basic IMPLEMENTS I_NovRamDK
VAR
//**********************************
// Static variables
//**********************************
	_bEnable: BOOL;
	_nDevId: UINT;
	_nMB_Offset: UINT;
	_nMB_Size: UINT;
//**********************************
// Methods variable
//**********************************
	FB_NovRamDK_M_nEnable_nMBSrc AT %MB0: BYTE;
	FB_NovRamDK_M_nEnable_nBank: BYTE;
	FB_NovRamDK_M_nEnable_nCalcSize: UINT;
	FB_NovRamDK_M_nEnable_iState: UINT;
	FB_NovRamDK_M_nEnable_fbExecute_R_TRIG: Tc2_Standard.R_TRIG;
	FB_NovRamDK_M_nEnable_fbExecute_F_TRIG: Tc2_Standard.F_TRIG;
	FB_NovRamDK_M_nEnable_fbGetDPRAMInfo: Tc2_IoFunctions.FB_GetDPRAMInfo;
	FB_NovRamDK_M_nEnable_stNovRamAddrInfo: Tc2_IoFunctions.ST_NovRamAddrInfo;
	FB_NovRamDK_M_nEnable_nArrStatus: ARRAY[1..5] OF UDINT;

	FB_NovRamDK_M_nRead_fbNovRamReadWriteEx: FB_NovRamReadWriteEx;
	FB_NovRamDK_M_nRead_iState: UINT;
	FB_NovRamDK_M_nRead_nBank: BYTE;

	FB_NovRamDK_M_nWrite_fbNovRamReadWriteEx: FB_NovRamReadWriteEx;
	FB_NovRamDK_M_nWrite_bReady: BOOL;
	FB_NovRamDK_M_nWrite_iState: UINT;
	FB_NovRamDK_M_nWrite_nBank: BYTE;
	FB_NovRamDK_M_nWrite_pByte: POINTER TO BYTE;
	FB_NovRamDK_M_nWrite_pCard: POINTER TO BYTE;
END_VAR

//	The result of the method is an unsigned double integer
//	0 = idle 
//	1 = coupled
//	2 = starting
//	3 = running
//	4 = aborted
// 	5 = no hardware connected
// 	6 = spare
//	7 = pointer or index error
//	8 = mapping error
//	9 = parameter error
//	10 = complete
//	Any other number = ErrorID
METHOD PUBLIC M_nEnable : UDINT
VAR_INPUT
	bExecute: BOOL;
	nDevId: UINT;
	nMB_Offset: UINT;
	nMB_Size: UINT;
END_VAR
//**********************************
// Local variable
//**********************************
THIS^._bEnable:= bExecute;
THIS^._nDevId:= nDevId;
THIS^._nMB_Offset:= nMB_Offset;
THIS^._nMB_Size:= nMB_Size;

//**********************************
// Reset
//**********************************
IF _bReset THEN
	IF _bError THEN
		FB_NovRamDK_M_nEnable_iState:= 000;
	END_IF
	M_nReset(bExecute:= _bReset);
END_IF

//**********************************
// Wait for execute
//**********************************
FB_NovRamDK_M_nEnable_fbExecute_R_TRIG(CLK:= bExecute);
FB_NovRamDK_M_nEnable_fbExecute_F_TRIG(CLK:= bExecute);
IF FB_NovRamDK_M_nEnable_fbExecute_R_TRIG.Q OR FB_NovRamDK_M_nEnable_fbExecute_F_TRIG.Q THEN
	FB_NovRamDK_M_nEnable_iState:= 000;
END_IF


//**********************************
// State maschine
//**********************************
CASE FB_NovRamDK_M_nEnable_iState OF
	
	000:	// Init
			M_nEnable:= cSTARTING;	
			_bReady:= FALSE; 
			FB_NovRamDK_M_nEnable_fbGetDPRAMInfo(bExecute:= FALSE); 
			IF M_nRead(bExecute:= FALSE) = cIDLE AND M_nWrite(bExecute:= FALSE) = cIDLE THEN
				FB_NovRamDK_M_nEnable_iState:= FB_NovRamDK_M_nEnable_iState +1;
			END_IF
	
	001:	// Wait for execute 
			M_nEnable:= cRUNNING;	
			IF bExecute THEN
				FB_NovRamDK_M_nEnable_iState:= FB_NovRamDK_M_nEnable_iState +1;
			END_IF
		
	002:	// Check parameter	
			M_nEnable:= cRUNNING;	
			IF _nDevId > 0 AND (nMB_Offset MOD 4 = 0) AND _nMB_Size > 0 AND (_nMB_Size MOD 4 = 0) THEN
				FB_NovRamDK_M_nEnable_iState:= FB_NovRamDK_M_nEnable_iState +1;
			ELSE
				M_nEnable:= cPARAMETER_ERROR;	
			END_IF	
		
	003:	// Calculate NovRam Size for ARM cpu
			M_nEnable:= cRUNNING;	
			IF (_nMB_Size + nMB_Offset) MOD 4 = 0 THEN
				FB_NovRamDK_M_nEnable_nCalcSize:= (_nMB_Size + nMB_Offset);
			ELSE
				FB_NovRamDK_M_nEnable_nCalcSize:= ((_nMB_Size + nMB_Offset) - (_nMB_Size + nMB_Offset MOD 4))+ 4;
			END_IF
			FB_NovRamDK_M_nEnable_iState:= FB_NovRamDK_M_nEnable_iState +1;
		
	004:	// Read NovRam size 
			M_nEnable:= cRUNNING;	
			FB_NovRamDK_M_nEnable_fbGetDPRAMInfo(
				nDevId:= _nDevId, 
				bExecute:= TRUE, 
				tTimeOut:= Tc2_System.DEFAULT_ADS_TIMEOUT, 
				bBusy=> , 
				bError=> , 
				nErrid=> , 
				stInfo=> FB_NovRamDK_M_nEnable_stNovRamAddrInfo);
	
			// Error
			IF FB_NovRamDK_M_nEnable_fbGetDPRAMInfo.bError THEN
				M_nError(nErrorID:= FB_NovRamDK_M_nEnable_fbGetDPRAMInfo.nErrId);
				M_nEnable:= FB_NovRamDK_M_nEnable_fbGetDPRAMInfo.nErrId;
			ELSE
				// Done
				IF NOT FB_NovRamDK_M_nEnable_fbGetDPRAMInfo.bBusy THEN
					FB_NovRamDK_M_nEnable_fbGetDPRAMInfo(bExecute:= FALSE); 
					FB_NovRamDK_M_nEnable_iState:= FB_NovRamDK_M_nEnable_iState +1;
				END_IF
			END_IF	
		
	005:	// Check max NovRam size
			M_nEnable:= cRUNNING;	
			IF FB_NovRamDK_M_nEnable_nCalcSize > ((FB_NovRamDK_M_nEnable_stNovRamAddrInfo.iCardMemSize/2) - 2) THEN
				FB_NovRamDK_M_nEnable_nCalcSize:= UDINT_TO_UINT(FB_NovRamDK_M_nEnable_stNovRamAddrInfo.iCardMemSize/2);
				FB_NovRamDK_M_nEnable_nCalcSize:= FB_NovRamDK_M_nEnable_nCalcSize - 4;
			END_IF
			FB_NovRamDK_M_nEnable_iState:= FB_NovRamDK_M_nEnable_iState +1;
	
	006:	// Read
			M_nEnable:= cRUNNING;	
			FB_NovRamDK_M_nEnable_nArrStatus[1]:= M_nRead(bExecute:= TRUE);
	
			// Error
			IF FB_NovRamDK_M_nEnable_nArrStatus[1] > cCOMPLETE THEN
				M_nError(nErrorID:= FB_NovRamDK_M_nEnable_nArrStatus[1]);
				M_nEnable:= FB_NovRamDK_M_nEnable_nArrStatus[1];
			ELSE
				// Done
				IF FB_NovRamDK_M_nEnable_nArrStatus[1] = cCOMPLETE THEN
					M_nRead(bExecute:= FALSE);
					FB_NovRamDK_M_nEnable_iState:= FB_NovRamDK_M_nEnable_iState +1;
				END_IF
			END_IF
			
	007:	// Write
			M_nEnable:= cRUNNING;	
			FB_NovRamDK_M_nEnable_nArrStatus[2]:= M_nWrite(bExecute:= TRUE);
			
			// Error
			IF FB_NovRamDK_M_nEnable_nArrStatus[2] > cCOMPLETE THEN
				M_nError(nErrorID:= FB_NovRamDK_M_nEnable_nArrStatus[2]);
				M_nEnable:= FB_NovRamDK_M_nEnable_nArrStatus[2];
			ELSE
				// Done
				IF FB_NovRamDK_M_nEnable_nArrStatus[2] = cCOMPLETE THEN
					M_nWrite(bExecute:= FALSE);
					FB_NovRamDK_M_nEnable_iState:= FB_NovRamDK_M_nEnable_iState +1;
				END_IF
			END_IF
	
	008:	// Done
			M_nEnable:= cCOMPLETE;	
			M_nWrite(bExecute:= TRUE);
			_bReady:= TRUE; 

ELSE
	FB_NovRamDK_M_nEnable_iState:= 000;
END_CASE
END_METHOD

//	The result of the method is an unsigned double integer
//	0 = idle 
//	1 = coupled
//	2 = starting
//	3 = running
//	4 = aborted
// 	5 = no hardware connected
// 	6 = spare
//	7 = pointer or index error
//	8 = mapping error
//	9 = parameter error
//	10 = complete
//	Any other number = ErrorID
METHOD PRIVATE M_nRead : UDINT
VAR_INPUT
	bExecute: BOOL;
END_VAR
//**********************************
// Reset
//**********************************
IF _bReset THEN
	IF _bError THEN
		FB_NovRamDK_M_nRead_iState:= 000;
	END_IF
END_IF


//**********************************
// State maschine 
//**********************************
CASE FB_NovRamDK_M_nRead_iState OF

	000: 	// Init 
			M_nRead:= cSTARTING;
			FB_NovRamDK_M_nRead_fbNovRamReadWriteEx(bRead:= FALSE, bWrite:= FALSE);
			FB_NovRamDK_M_nRead_iState:= FB_NovRamDK_M_nRead_iState +1;

	001:	// Wait for execute 
			M_nRead:= cIDLE;
			IF bExecute THEN
				FB_NovRamDK_M_nRead_iState:= FB_NovRamDK_M_nRead_iState +1;
			END_IF

	002:	// Read databank value 
			M_nRead:= cRUNNING;
			FB_NovRamDK_M_nRead_fbNovRamReadWriteEx(
				nDevId:= _nDevId,
				bRead:= TRUE,
				bWrite:= FALSE,
				cbSrcLen:= 1,
				cbDestLen:= 1,
				pSrcAddr:= ADR(FB_NovRamDK_M_nRead_nBank),
				pDestAddr:= ADR(FB_NovRamDK_M_nRead_nBank),
				nReadOffs:= FB_NovRamDK_M_nEnable_stNovRamAddrInfo.iCardMemSize -1,
				nWriteOffs:= 0,
				tTimeOut:= T#2s,
				bBusy=> ,
				bError=> ,
				nErrId=> ,
				cbRead=> ,
				cbWrite=> );
	
			// Error	
			IF FB_NovRamDK_M_nRead_fbNovRamReadWriteEx.bError THEN
				M_nError(nErrorID:= FB_NovRamDK_M_nRead_fbNovRamReadWriteEx.nErrId);
				M_nRead:= FB_NovRamDK_M_nRead_fbNovRamReadWriteEx.nErrId;
			ELSE
				// Done
				IF NOT FB_NovRamDK_M_nRead_fbNovRamReadWriteEx.bBusy AND FB_NovRamDK_M_nRead_fbNovRamReadWriteEx.cbRead = 1 THEN
					FB_NovRamDK_M_nRead_fbNovRamReadWriteEx(bRead:= FALSE,	bWrite:= FALSE);
					FB_NovRamDK_M_nRead_iState:= FB_NovRamDK_M_nRead_iState +1;
				END_IF
			END_IF
	
	003:	// ReadNovRam data from databank 0 or 1 
			M_nRead:= cRUNNING;
			IF FB_NovRamDK_M_nRead_nBank = 0 THEN
				FB_NovRamDK_M_nRead_fbNovRamReadWriteEx(
					nDevId:= _nDevId,
					bRead:= TRUE,
					bWrite:= FALSE,
					cbSrcLen:= FB_NovRamDK_M_nEnable_nCalcSize,
					cbDestLen:= FB_NovRamDK_M_nEnable_nCalcSize,
					pSrcAddr:= ADR(FB_NovRamDK_M_nEnable_nMBSrc),
					pDestAddr:= ADR(FB_NovRamDK_M_nEnable_nMBSrc),
					nReadOffs:= 0,
					nWriteOffs:= 0,
					tTimeOut:= T#2s,
					bBusy=> ,
					bError=> ,
					nErrId=> ,
					cbRead=> ,
					cbWrite=> );
			ELSE
				FB_NovRamDK_M_nRead_fbNovRamReadWriteEx(
					nDevId:= _nDevId,
					bRead:= TRUE,
					bWrite:= FALSE,
					cbSrcLen:= FB_NovRamDK_M_nEnable_nCalcSize,
					cbDestLen:= FB_NovRamDK_M_nEnable_nCalcSize,
					pSrcAddr:= ADR(FB_NovRamDK_M_nEnable_nMBSrc),
					pDestAddr:= ADR(FB_NovRamDK_M_nEnable_nMBSrc),
					nReadOffs:= FB_NovRamDK_M_nEnable_stNovRamAddrInfo.iCardMemSize / 2,
					nWriteOffs:= 0,
					tTimeOut:= T#2s,
					bBusy=> ,
					bError=> ,
					nErrId=> ,
					cbRead=> ,
					cbWrite=> );
			END_IF
	
			// Error	
			IF FB_NovRamDK_M_nRead_fbNovRamReadWriteEx.bError THEN
				M_nError(nErrorID:= FB_NovRamDK_M_nRead_fbNovRamReadWriteEx.nErrId);
				M_nRead:= FB_NovRamDK_M_nRead_fbNovRamReadWriteEx.nErrId;
			ELSE
				// Done
				IF NOT FB_NovRamDK_M_nRead_fbNovRamReadWriteEx.bBusy AND FB_NovRamDK_M_nRead_fbNovRamReadWriteEx.cbRead = FB_NovRamDK_M_nEnable_nCalcSize THEN
					FB_NovRamDK_M_nRead_fbNovRamReadWriteEx(bRead:= FALSE,	bWrite:= FALSE);
					FB_NovRamDK_M_nRead_iState:= FB_NovRamDK_M_nRead_iState +1;
				END_IF
			END_IF
	
	004:	// Read done 
			M_nRead:= cCOMPLETE;
			IF NOT bExecute THEN
				FB_NovRamDK_M_nRead_iState:= 000;
			END_IF

ELSE
	FB_NovRamDK_M_nRead_iState:= 000;
END_CASE
END_METHOD

//	The result of the method is an unsigned double integer
//	0 = idle 
//	1 = coupled
//	2 = starting
//	3 = running
//	4 = aborted
// 	5 = no hardware connected
// 	6 = spare
//	7 = pointer or index error
//	8 = mapping error
//	9 = parameter error
//	10 = complete
//	Any other number = ErrorID
METHOD PRIVATE M_nWrite : UDINT
VAR_INPUT
	bExecute: BOOL;
END_VAR
//**********************************
// Reset
//**********************************
IF _bReset THEN
	IF _bError THEN
		FB_NovRamDK_M_nWrite_iState:= 000;
	END_IF
END_IF


//**********************************
// State maschine 
//**********************************
CASE FB_NovRamDK_M_nWrite_iState OF

	000:	// Init
			M_nWrite:= cSTARTING;
			FB_NovRamDK_M_nWrite_fbNovRamReadWriteEx(bRead:= FALSE,	bWrite:= FALSE);
			FB_NovRamDK_M_nWrite_bReady:= FALSE;
			FB_NovRamDK_M_nWrite_iState:= FB_NovRamDK_M_nWrite_iState +1;

	001:	// Wait for execute 
			M_nWrite:= cIDLE;
			IF bExecute THEN
				FB_NovRamDK_M_nWrite_iState:= FB_NovRamDK_M_nWrite_iState +1;
			END_IF

	002:	// Read databank value 
			M_nWrite:= cRUNNING;
			FB_NovRamDK_M_nWrite_fbNovRamReadWriteEx(
				nDevId:= _nDevId,
				bRead:= TRUE,
				bWrite:= FALSE,
				cbSrcLen:= 1,
				cbDestLen:= 1,
				pSrcAddr:= ADR(FB_NovRamDK_M_nWrite_nBank),
				pDestAddr:= ADR(FB_NovRamDK_M_nWrite_nBank),
				nReadOffs:= FB_NovRamDK_M_nEnable_stNovRamAddrInfo.iCardMemSize -1,
				nWriteOffs:= 0,
				tTimeOut:= T#2s,
				bBusy=> ,
				bError=> ,
				nErrId=> ,
				cbRead=> ,
				cbWrite=> );
	
			// Error
			IF FB_NovRamDK_M_nWrite_fbNovRamReadWriteEx.bError THEN
				M_nError(nErrorID:= FB_NovRamDK_M_nWrite_fbNovRamReadWriteEx.nErrId);
				M_nWrite:= FB_NovRamDK_M_nWrite_fbNovRamReadWriteEx.nErrId;
			ELSE	
				// Done				
				IF FB_NovRamDK_M_nWrite_fbNovRamReadWriteEx.cbRead = 1 THEN
					FB_NovRamDK_M_nWrite_fbNovRamReadWriteEx(bRead:= FALSE,	bWrite:= FALSE);
					FB_NovRamDK_M_nWrite_iState:= FB_NovRamDK_M_nWrite_iState +1;
				END_IF
			END_IF
		
	003:	// Pointer settings 
			M_nWrite:= cRUNNING;
			FB_NovRamDK_M_nWrite_pByte:= ADR(FB_NovRamDK_M_nWrite_nBank);
			FB_NovRamDK_M_nWrite_pCard:= FB_NovRamDK_M_nEnable_stNovRamAddrInfo.pCardAddress + FB_NovRamDK_M_nEnable_stNovRamAddrInfo.iCardMemSize -1;
			FB_NovRamDK_M_nWrite_iState:= FB_NovRamDK_M_nWrite_iState +1;
		
	004:	// Write ready 
			M_nWrite:= cCOMPLETE;
			FB_NovRamDK_M_nWrite_bReady:= TRUE;
			IF NOT bExecute THEN
				FB_NovRamDK_M_nWrite_iState:= 000;
			END_IF
		
ELSE
	FB_NovRamDK_M_nWrite_iState:= 000;
END_CASE


// Write data to databank 0 or 1 
IF bExecute AND FB_NovRamDK_M_nWrite_bReady THEN
	IF FB_NovRamDK_M_nWrite_nBank = 1 THEN
		FB_NovRamDK_M_nWrite_nBank:= 0;
		Tc2_System.MEMCPY(destAddr:= FB_NovRamDK_M_nEnable_stNovRamAddrInfo.pCardAddress, srcAddr:= ADR(FB_NovRamDK_M_nEnable_nMBSrc) + _nMB_Offset, n:= FB_NovRamDK_M_nEnable_nCalcSize);
		FB_NovRamDK_M_nWrite_pCard^:= FB_NovRamDK_M_nWrite_pByte^;
	ELSE
		FB_NovRamDK_M_nWrite_nBank:= 1;
		Tc2_System.MEMCPY(destAddr:= FB_NovRamDK_M_nEnable_stNovRamAddrInfo.pCardAddress + (FB_NovRamDK_M_nEnable_stNovRamAddrInfo.iCardMemSize/2), srcAddr:= ADR(FB_NovRamDK_M_nEnable_nMBSrc) + _nMB_Offset, n:= FB_NovRamDK_M_nEnable_nCalcSize);
		FB_NovRamDK_M_nWrite_pCard^:= FB_NovRamDK_M_nWrite_pByte^;
	END_IF
END_IF
END_METHOD

END_FUNCTION_BLOCK

// POUs/SYSTEM/FBs/Persistent/ITFs/I_WritePersistentDataDK
INTERFACE I_WritePersistentDataDK EXTENDS I_Basic

//	The result of the method is an unsigned double integer
//	0 = idle 
//	1 = coupled
//	2 = starting
//	3 = running
//	4 = aborted
// 	5 = no hardware connected
//  6 = Spare
//	7 = pointer or index error
//	8 = mapping error
//	9 = parameter error
//	10 = complete
//	Any other number = ErrorID
METHOD PUBLIC M_n1_Second_UPS : UDINT
VAR_INPUT
	bExecute: BOOL;
END_VAR
END_METHOD

//	The result of the method is an unsigned double integer
//	0 = idle 
//	1 = coupled
//	2 = starting
//	3 = running
//	4 = aborted
// 	5 = no hardware connected
//  6 = Spare
//	7 = pointer or index error
//	8 = mapping error
//	9 = parameter error
//	10 = complete
//	Any other number = ErrorID
METHOD M_nEnable : UDINT
VAR_INPUT
	bExecute: BOOL;
	tLogTimePuls: TIME;
END_VAR
END_METHOD

//	The result of the method is an unsigned double integer
//	0 = idle 
//	1 = coupled
//	2 = starting
//	3 = running
//	4 = aborted
// 	5 = no hardware connected
//  6 = Spare
//	7 = pointer or index error
//	8 = mapping error
//	9 = parameter error
//	10 = complete
//	Any other number = ErrorID
METHOD M_nWrite : UDINT
VAR_INPUT
	bExecute: BOOL;
END_VAR
END_METHOD

PROPERTY PUBLIC P_bBusy : BOOL
GET
END_GET
END_PROPERTY

PROPERTY PUBLIC P_bPowerFailDetect : BOOL
GET
END_GET
END_PROPERTY

PROPERTY PUBLIC P_ePersistentMode  : E_PersistentMode
SET
END_SET
END_PROPERTY

PROPERTY PUBLIC P_eSUPS_Mode : Tc2_SUPS.E_S_UPS_Mode
SET
END_SET
END_PROPERTY

PROPERTY PUBLIC P_nWriteCNT : UDINT
GET
END_GET
END_PROPERTY

END_INTERFACE

// POUs/SYSTEM/FBs/Persistent/FB_WritePersistentDataDK
//------------------------------------------------------------------------------------------
//                                                                                        	
//***************************** Beckhoff TwinCAT Examples **********************************
//                                                                                        	
//************************************* WARNING ********************************************
// This program is only an example. If it is used as a control program in any real        	
// application, Beckhoff is not responsible for any malfunction, loss or damage           	
// which could arise by using this program!                                               	
//                                                                                        	
//*************************************  Program Info. *************************************
//                                                                                        	
// PLC program name:       	FB_WritePersistentDataDK (FB)                                          	
// Hardware platform:      	TwinCat v3.1.4022				                          	
// Modified by:            	Hans Chr. Pallesen 			                                  	
// Email:					h.pallesen@beckhoff.com	                                  	
//                                                                                        	
// ======================================================================================== 
//         Version       Date                        Remarks                              	
// ======================================================================================== 
//         1.0           02 feb 2014                 First release of this example        	
// ======================================================================================== 
//                                                                                        	
//******************************* Aims OF this PLC PROGRAM *********************************
//                                                                                        	
// Write persistent data file				 			                                      	
//																	                      	
//                                                                                        	
//----------------------------------------------------------------------------------------- 
FUNCTION_BLOCK FB_WritePersistentDataDK EXTENDS FB_Basic IMPLEMENTS I_WritePersistentDataDK
VAR
//**************************
// Static variables
//**************************
	_bFirstBoot: BOOL := TRUE;
	_nAdsPort: UINT;
	_bPowerFailDetect: BOOL;
	_b1Sec_UPS_Pressent: BOOL;
	_fbWritePersistentData: Tc2_Utilities.FB_WritePersistentData;
	
//**************************
// Property variables
//**************************
	_bBusy: BOOL;	
	_nWriteCNT: UDINT;
	_eUpsMode: Tc2_SUPS.E_S_UPS_Mode:= E_S_UPS_Mode.eSUPS_WrPersistData_Shutdown;
	_ePersistentMode: Tc2_Utilities.E_PersistentMode:= E_PersistentMode.SPDM_2PASS;
	
//**************************
// Methods variable
//**************************

	FB_WritePersistentDataDK_M_nEnable_iState: INT;
	FB_WritePersistentDataDK_M_nEnable_fbExecute_R_TRIG: R_TRIG;
	FB_WritePersistentDataDK_M_nEnable_fbReset_R_TRIG: R_TRIG;
	FB_WritePersistentDataDK_M_nEnable_fbStartDelay_TON: TON;
	FB_WritePersistentDataDK_M_nEnable_fbLogTimePuls_TON: TON;
	
	FB_WritePersistentDataDK_M_nWrite_iState: INT;
	FB_WritePersistentDataDK_M_nWrite_fbExecute_R_TRIG: R_TRIG;
	FB_WritePersistentDataDK_M_nWrite_fbReset_R_TRIG: R_TRIG;
	
	FB_WritePersistentDataDK_M_n1_Second_UPS_iState: INT;
	FB_WritePersistentDataDK_M_n1_Second_UPS_bReady: BOOL;
	FB_WritePersistentDataDK_M_n1_Second_UPS_stDeviceIdentificationEx: Tc2_Utilities.ST_DeviceIdentificationEx;
	FB_WritePersistentDataDK_M_n1_Second_UPS_fb_GetDeviceIdentificationEx: Tc2_Utilities.FB_GetDeviceIdentificationEx;
	FB_WritePersistentDataDK_M_n1_Second_UPS_fbGetUPSStatus: Tc2_IoFunctions.FB_GetUPSStatus;
	FB_WritePersistentDataDK_M_n1_Second_UPS_fbS_UPS_BAPI : Tc2_SUPS.FB_S_UPS_BAPI;
	FB_WritePersistentDataDK_M_n1_Second_UPS_fbDelay_TON: Tc2_Standard.TON;
END_VAR

//	The result of the method is an unsigned double integer
//	0 = idle 
//	1 = coupled
//	2 = starting
//	3 = running
//	4 = aborted
// 	5 = no hardware connected
// 	6 = spare
//	7 = pointer or index error
//	8 = mapping error
//	9 = parameter error
//	10 = complete
//	Any other number = ErrorID
METHOD PUBLIC M_n1_Second_UPS : UDINT
VAR_INPUT
	bExecute: BOOL;
END_VAR
_bPowerFailDetect:= FALSE;
IF FB_WritePersistentDataDK_M_n1_Second_UPS_bReady THEN
	IF _b1Sec_UPS_Pressent THEN

		// Update 1sec UPS device
		FB_WritePersistentDataDK_M_n1_Second_UPS_fbS_UPS_BAPI(
			sNetID:= , 
			iPLCPort:= _nAdsPort, 
			tTimeout:= , 
			eUpsMode:= _eUpsMode, 
			ePersistentMode:= _ePersistentMode, 
			tRecoverTime:= , 
			bPowerFailDetect=> _bPowerFailDetect, 
			eState=> , 
			nCapacity=> , 
			bBusy=> , 
			bError=> , 
			nErrID=> );

	ELSE
	
		// Update any UPS device
		FB_WritePersistentDataDK_M_n1_Second_UPS_fbGetUPSStatus(
			sNetId:= , 
			nPort:= 0, 
			bEnable:= TRUE, 
			bValid=> , 
			bError=> , 
			nErrId=> , 
			stStatus=> );
		
		IF FB_WritePersistentDataDK_M_n1_Second_UPS_fbGetUPSStatus.bValid THEN
			IF FB_WritePersistentDataDK_M_n1_Second_UPS_fbGetUPSStatus.stStatus.ePowerStatus = Tc2_IoFunctions.PowerOnBattery THEN
				_bPowerFailDetect:= TRUE;	
			END_IF
		END_IF	
	
	END_IF
	
END_IF

	
//**********************************
// Reset 
//**********************************
IF _bReset THEN
	IF _bError THEN	
		FB_WritePersistentDataDK_M_n1_Second_UPS_iState:= 000;
	END_IF	
END_IF


//**********************************
// State maschine
//**********************************
CASE FB_WritePersistentDataDK_M_n1_Second_UPS_iState OF
	
	000:	// Wait for execute and start delay
			M_n1_Second_UPS:= cIDLE;
			FB_WritePersistentDataDK_M_n1_Second_UPS_fbGetUPSStatus(bEnable:= FALSE); 
			FB_WritePersistentDataDK_M_n1_Second_UPS_bReady:= FALSE;
			FB_WritePersistentDataDK_M_n1_Second_UPS_fbDelay_TON(IN:= FALSE, PT:= , Q=> , ET=> );
			IF bExecute THEN
				FB_WritePersistentDataDK_M_n1_Second_UPS_iState:= FB_WritePersistentDataDK_M_n1_Second_UPS_iState +1;
			END_IF	

	001:	// Get data	
			M_n1_Second_UPS:= cRUNNING;
			FB_WritePersistentDataDK_M_n1_Second_UPS_fb_GetDeviceIdentificationEx(bExecute:= FALSE); 
			FB_WritePersistentDataDK_M_n1_Second_UPS_fb_GetDeviceIdentificationEx(
				bExecute:= TRUE, 
				tTimeout:= Tc2_System.DEFAULT_ADS_TIMEOUT, 
				sNetId:= '', 
				bBusy=> , 
				bError=> , 
				nErrorID=> , 
				stDevIdent=> FB_WritePersistentDataDK_M_n1_Second_UPS_stDeviceIdentificationEx);
	
			FB_WritePersistentDataDK_M_n1_Second_UPS_iState:= FB_WritePersistentDataDK_M_n1_Second_UPS_iState +1;
	
	002:	// Get data done
			M_n1_Second_UPS:= cRUNNING;
			FB_WritePersistentDataDK_M_n1_Second_UPS_fb_GetDeviceIdentificationEx(bExecute:= FALSE, stDevIdent=> FB_WritePersistentDataDK_M_n1_Second_UPS_stDeviceIdentificationEx);
			IF FB_WritePersistentDataDK_M_n1_Second_UPS_fb_GetDeviceIdentificationEx.bError THEN
				M_nError(nErrorID:= FB_WritePersistentDataDK_M_n1_Second_UPS_fb_GetDeviceIdentificationEx.nErrorID);
				M_n1_Second_UPS:= FB_WritePersistentDataDK_M_n1_Second_UPS_fb_GetDeviceIdentificationEx.nErrorID;
			ELSE
				// Done
				IF NOT FB_WritePersistentDataDK_M_n1_Second_UPS_fb_GetDeviceIdentificationEx.bBusy THEN
					FB_WritePersistentDataDK_M_n1_Second_UPS_iState:= FB_WritePersistentDataDK_M_n1_Second_UPS_iState +1;
				END_IF	
			END_IF
		
	003:	// Check 1sec UPS device pressent
			M_n1_Second_UPS:= cRUNNING;
			FB_WritePersistentDataDK_M_n1_Second_UPS_fbDelay_TON(IN:= TRUE, PT:= T#1S, Q=> , ET=> );
			
			// Update UPS 1sec device
			FB_WritePersistentDataDK_M_n1_Second_UPS_fbS_UPS_BAPI(
				sNetID:= , 
				iPLCPort:= , 
				tTimeout:= , 
				eUpsMode:= _eUpsMode, 
				ePersistentMode:= _ePersistentMode, 
				tRecoverTime:= , 
				bPowerFailDetect=> , 
				eState=> , 
				nCapacity=> , 
				bBusy=> , 
				bError=> , 
				nErrID=> );
			
			// 1sec UPS device pressent			
			IF FB_WritePersistentDataDK_M_n1_Second_UPS_fbDelay_TON.Q THEN
				_b1Sec_UPS_Pressent:= TRUE;
				IF FB_WritePersistentDataDK_M_n1_Second_UPS_fbS_UPS_BAPI.bError THEN
					_b1Sec_UPS_Pressent:= FALSE;
				END_IF
				IF FB_WritePersistentDataDK_M_n1_Second_UPS_fbS_UPS_BAPI.nErrID > 0000 THEN
					_b1Sec_UPS_Pressent:= FALSE;
				END_IF
				FB_WritePersistentDataDK_M_n1_Second_UPS_iState:= FB_WritePersistentDataDK_M_n1_Second_UPS_iState +1;
			END_IF

	004:	// Check UPS hardware connected	
			M_n1_Second_UPS:= cRUNNING;
			FB_WritePersistentDataDK_M_n1_Second_UPS_bReady:= TRUE;
			IF bExecute THEN
				IF _b1Sec_UPS_Pressent THEN
					M_n1_Second_UPS:= cCOMPLETE;
				ELSE
					M_n1_Second_UPS:= cNO_HARDWARE_CONNECTED;
				END_IF
			ELSE
				FB_WritePersistentDataDK_M_n1_Second_UPS_iState:= 000;
			END_IF	

ELSE
	FB_WritePersistentDataDK_M_n1_Second_UPS_iState:= 000;
END_CASE
END_METHOD

//	The result of the method is an unsigned double integer
//	0 = idle 
//	1 = coupled
//	2 = starting
//	3 = running
//	4 = aborted
// 	5 = no hardware connected
// 	6 = spare
//	7 = pointer or index error
//	8 = mapping error
//	9 = parameter error
//	10 = complete
//	Any other number = ErrorID
METHOD PUBLIC M_nEnable : UDINT
VAR_INPUT
	bExecute: BOOL;
	tLogTimePuls: TIME;
END_VAR
// Local variable
THIS^._nAdsPort:= TwinCAT_SystemInfoVarList._AppInfo.AdsPort;

//**********************************
// Reset 
//**********************************
IF _bReset THEN
	IF _bError THEN	
		FB_WritePersistentDataDK_M_nEnable_iState:= 000;
	END_IF	
	M_nReset(bExecute:= _bReset);
END_IF

// Power fail
FB_WritePersistentDataDK_M_nEnable_fbReset_R_TRIG(CLK:= _bPowerFailDetect, Q=> );
IF FB_WritePersistentDataDK_M_nEnable_fbReset_R_TRIG.Q THEN
	IF _b1Sec_UPS_Pressent THEN
		FB_WritePersistentDataDK_M_nEnable_iState:= 000;
	ELSE
		FB_WritePersistentDataDK_M_nEnable_iState:= 001;
	END_IF
END_IF

// Startup delay
FB_WritePersistentDataDK_M_nEnable_fbStartDelay_TON(IN:= TRUE, PT:= T#15S);

// LogTtime puls
IF FB_WritePersistentDataDK_M_nEnable_fbStartDelay_TON.Q THEN
	FB_WritePersistentDataDK_M_nEnable_fbLogTimePuls_TON(IN:= bExecute AND tLogTimePuls > T#0MS AND NOT FB_WritePersistentDataDK_M_nEnable_fbLogTimePuls_TON.Q AND NOT _bPowerFailDetect, PT:= tLogTimePuls);
ELSE
	FB_WritePersistentDataDK_M_nEnable_fbLogTimePuls_TON(IN:= FALSE);
END_IF	

//**********************************
// Wait for execute
//**********************************
IF FB_WritePersistentDataDK_M_nEnable_fbStartDelay_TON.Q THEN
	FB_WritePersistentDataDK_M_nEnable_fbExecute_R_TRIG(CLK:= (_bFirstBoot OR FB_WritePersistentDataDK_M_nEnable_fbLogTimePuls_TON.Q) AND NOT _bPowerFailDetect);
	IF FB_WritePersistentDataDK_M_nEnable_fbExecute_R_TRIG.Q THEN
		FB_WritePersistentDataDK_M_nEnable_iState:= 001;
	END_IF
ELSE
	FB_WritePersistentDataDK_M_nEnable_fbExecute_R_TRIG(CLK:= FALSE);
	FB_WritePersistentDataDK_M_nEnable_iState:= 000;
END_IF


//**********************************
// Main sekvens
//**********************************
CASE FB_WritePersistentDataDK_M_nEnable_iState OF

	000:	// Do nothing
			M_nEnable:= cIDLE;
			IF _bError THEN
				M_nEnable:= _nErrorID;
			ELSE
				IF bExecute THEN
					IF FB_WritePersistentDataDK_M_nEnable_fbStartDelay_TON.Q THEN
						M_nEnable:= cCOMPLETE;
					ELSE
						M_nEnable:= cSTARTING;
					END_IF
				END_IF	
			END_IF

	001:	// Init
			M_nEnable:= cSTARTING;
			_fbWritePersistentData.PORT:= _nAdsPort;
			_fbWritePersistentData.MODE:= _ePersistentMode;
			_fbWritePersistentData.TMOUT:= Tc2_System.DEFAULT_ADS_TIMEOUT;
			FB_WritePersistentDataDK_M_nEnable_iState:= FB_WritePersistentDataDK_M_nEnable_iState +1;

	002:	// Running
			M_nEnable:= cRUNNING;
			IF _fbWritePersistentData.BUSY THEN
				FB_WritePersistentDataDK_M_nEnable_iState:= FB_WritePersistentDataDK_M_nEnable_iState +3;
			ELSE
				FB_WritePersistentDataDK_M_nEnable_iState:= FB_WritePersistentDataDK_M_nEnable_iState +1;
			END_IF
			
	003:	// Init
			M_nEnable:= cRUNNING;
			_fbWritePersistentData.START:= FALSE; 
			FB_WritePersistentDataDK_M_nEnable_iState:= FB_WritePersistentDataDK_M_nEnable_iState +1;

	004:	// Start
			M_nEnable:= cRUNNING;
			_fbWritePersistentData.START:= TRUE; 
			FB_WritePersistentDataDK_M_nEnable_iState:= FB_WritePersistentDataDK_M_nEnable_iState +1;

	005:	// Write persistent data - Done
			M_nEnable:= cRUNNING;
		
			// Error handling
			IF _fbWritePersistentData.ERR THEN
				M_nError(nErrorID:= _fbWritePersistentData.ERRID);	
				M_nEnable:= _fbWritePersistentData.ERRID;
			ELSE
				// Done
				IF NOT _fbWritePersistentData.BUSY THEN
					IF _bFirstBoot THEN
						_fbWritePersistentData.START:= FALSE; 
						FB_WritePersistentDataDK_M_nEnable_iState:= FB_WritePersistentDataDK_M_nEnable_iState +1;
					ELSE
						_nWriteCNT:= _nWriteCNT +1;
						_fbWritePersistentData.START:= FALSE; 
						FB_WritePersistentDataDK_M_nEnable_iState:= 100;
					END_IF
				END_IF	
			END_IF

	006:	// Init
			M_nEnable:= cSTARTING;
			_fbWritePersistentData.START:= FALSE; 
			FB_WritePersistentDataDK_M_nEnable_iState:= FB_WritePersistentDataDK_M_nEnable_iState +1;

	007:	// Start
			M_nEnable:= cRUNNING;
			_fbWritePersistentData.START:= TRUE; 
			FB_WritePersistentDataDK_M_nEnable_iState:= FB_WritePersistentDataDK_M_nEnable_iState +1;
			
	008:	// Write persistent data - Done
			M_nEnable:= cRUNNING;
		
			// Error handling
			IF _fbWritePersistentData.ERR THEN
				M_nError(nErrorID:= _fbWritePersistentData.ERRID);	
				M_nEnable:= _fbWritePersistentData.ERRID;
			ELSE
				// Done
				IF NOT _fbWritePersistentData.BUSY THEN
					_nWriteCNT:= _nWriteCNT +1;
					_fbWritePersistentData.START:= FALSE; 
					FB_WritePersistentDataDK_M_nEnable_iState:= 100;
				END_IF	
			END_IF
	
	100:	// Done
			M_nEnable:= cCOMPLETE;
			_bFirstBoot:= FALSE;
			FB_WritePersistentDataDK_M_nEnable_iState:= 000;

ELSE
	FB_WritePersistentDataDK_M_nEnable_iState:= 000;	
END_CASE


// Proporty update
IF NOT _bError AND FB_WritePersistentDataDK_M_nEnable_fbStartDelay_TON.Q AND NOT _bPowerFailDetect THEN
	_bReady:= TRUE; 
ELSE
	_bReady:= FALSE; 
END_IF

// Status update
_fbWritePersistentData(TMOUT:= T#30S); 
_bBusy:= _fbWritePersistentData.BUSY;
END_METHOD

//	The result of the method is an unsigned double integer
//	0 = idle 
//	1 = coupled
//	2 = starting
//	3 = running
//	4 = aborted
// 	5 = no hardware connected
// 	6 = spare
//	7 = pointer or index error
//	8 = mapping error
//	9 = parameter error
//	10 = complete
//	Any other number = ErrorID
METHOD PUBLIC M_nWrite : UDINT
VAR_INPUT
	bExecute: BOOL;
END_VAR
//**********************************
// Reset 
//**********************************
IF _bReset THEN
	IF _bError THEN	
		FB_WritePersistentDataDK_M_nWrite_iState:= 000;
	END_IF	
END_IF

// Power fail
FB_WritePersistentDataDK_M_nWrite_fbReset_R_TRIG(CLK:= _bPowerFailDetect, Q=> );
IF FB_WritePersistentDataDK_M_nWrite_fbReset_R_TRIG.Q THEN
	FB_WritePersistentDataDK_M_nWrite_iState:= 000;
END_IF

//**********************************
// Wait for execute
//**********************************
IF _bReady THEN
	FB_WritePersistentDataDK_M_nWrite_fbExecute_R_TRIG(CLK:= bExecute AND NOT _bPowerFailDetect);
	IF FB_WritePersistentDataDK_M_nWrite_fbExecute_R_TRIG.Q THEN
		FB_WritePersistentDataDK_M_nWrite_iState:= 001;
	END_IF
ELSE
	FB_WritePersistentDataDK_M_nWrite_fbExecute_R_TRIG(CLK:= FALSE);
	FB_WritePersistentDataDK_M_nWrite_iState:= 000;
END_IF


//**********************************
// Main sekvens
//**********************************
CASE FB_WritePersistentDataDK_M_nWrite_iState OF

	000:	// Do nothing
	
	001:	// Running
			M_nWrite:= cRUNNING;
			IF _bBusy THEN
				FB_WritePersistentDataDK_M_nWrite_iState:= FB_WritePersistentDataDK_M_nWrite_iState +1;
			ELSE
				FB_WritePersistentDataDK_M_nWrite_iState:= FB_WritePersistentDataDK_M_nWrite_iState +2;
			END_IF

	002:	// Write persistent done
			M_nWrite:= cRUNNING;
			IF NOT _bBusy THEN
				_fbWritePersistentData.START:= FALSE; 
				FB_WritePersistentDataDK_M_nWrite_iState:= 100;
			END_IF
			
	003:	// Init
			M_nWrite:= cRUNNING;
			_fbWritePersistentData.START:= FALSE; 
			FB_WritePersistentDataDK_M_nWrite_iState:= FB_WritePersistentDataDK_M_nWrite_iState +1;

	004:	// Start
			M_nWrite:= cRUNNING;
			_fbWritePersistentData.START:= TRUE; 
			FB_WritePersistentDataDK_M_nWrite_iState:= FB_WritePersistentDataDK_M_nWrite_iState +1;

	005:	// Write persistent data - Done
			M_nWrite:= cRUNNING;
		
			// Error handling
			IF _fbWritePersistentData.ERR THEN
				M_nError(nErrorID:= _fbWritePersistentData.ERRID);	
				M_nWrite:= _fbWritePersistentData.ERRID;
			ELSE
				// Done
				IF NOT _bBusy THEN
					_nWriteCNT:= _nWriteCNT +1;
					_fbWritePersistentData.START:= FALSE; 	
					FB_WritePersistentDataDK_M_nWrite_iState:= 100;
				END_IF	
			END_IF
	
	100:	// Done
			M_nWrite:= cCOMPLETE;
			IF NOT bExecute THEN
				FB_WritePersistentDataDK_M_nWrite_iState:= 000;	
			END_IF	
	
ELSE
	FB_WritePersistentDataDK_M_nWrite_iState:= 000;	
END_CASE
END_METHOD

{attribute 'monitoring' := 'variable'}
PROPERTY PUBLIC P_bBusy : BOOL
GET
P_bBusy:= _bBusy;
END_GET
END_PROPERTY

{attribute 'monitoring' := 'variable'}
PROPERTY PUBLIC P_bPowerFailDetect : BOOL
GET
P_bPowerFailDetect:= _bPowerFailDetect;
END_GET
END_PROPERTY

{attribute 'monitoring' := 'variable'}
PROPERTY PUBLIC P_ePersistentMode  : E_PersistentMode
SET
_ePersistentMode:= P_ePersistentMode;
END_SET
END_PROPERTY

{attribute 'monitoring' := 'variable'}
PROPERTY PUBLIC P_eSUPS_Mode : Tc2_SUPS.E_S_UPS_Mode
SET
_eUpsMode:= P_eSUPS_Mode;
END_SET
END_PROPERTY

{attribute 'monitoring' := 'variable'}
PROPERTY PUBLIC P_nWriteCNT : UDINT
GET
P_nWriteCNT:= _nWriteCNT;
END_GET
END_PROPERTY

END_FUNCTION_BLOCK

// POUs/SYSTEM/FBs/System/ITFs/I_SystemDK
INTERFACE I_SystemDK EXTENDS I_Basic

//	The result of the method is an unsigned double integer
//	0 = idle 
//	1 = coupled
//	2 = starting
//	3 = running
//	4 = aborted
// 	5 = no hardware connected
//  6 = Spare
//	7 = pointer or index error
//	8 = mapping error
//	9 = parameter error
//	10 = complete
//	Any other number = ErrorID
METHOD PUBLIC M_nCerHost : UDINT
VAR_INPUT
	bEnable: BOOL;
	bDisable: BOOL;
END_VAR
END_METHOD

//	The result of the method is an unsigned double integer
//	0 = idle 
//	1 = coupled
//	2 = starting
//	3 = running
//	4 = aborted
// 	5 = no hardware connected
//  6 = Spare
//	7 = pointer or index error
//	8 = mapping error
//	9 = parameter error
//	10 = complete
//	Any other number = ErrorID
METHOD PUBLIC M_nEnable : UDINT
VAR_INPUT
END_VAR
END_METHOD

METHOD PUBLIC M_nGetTimeStampInMs : ULINT
VAR_INPUT
END_VAR
END_METHOD

PROPERTY PUBLIC P_bIs_ARM : BOOL
GET
END_GET
END_PROPERTY

PROPERTY PUBLIC P_bIs_CE_Device : BOOL
GET
END_GET
END_PROPERTY

PROPERTY PUBLIC P_bIs_x64 : BOOL
GET
END_GET
END_PROPERTY

PROPERTY PUBLIC P_bIs_x86 : BOOL
GET
END_GET
END_PROPERTY

PROPERTY PUBLIC P_nAdsPort : UINT
GET
END_GET
END_PROPERTY

PROPERTY PUBLIC P_nCycleTime : UDINT
GET
END_GET
END_PROPERTY

PROPERTY PUBLIC P_sHardwareSerialNumber : String
GET
END_GET
END_PROPERTY

PROPERTY PUBLIC P_stDeviceIdentificationEx : Tc2_Utilities.ST_DeviceIdentificationEx
GET
END_GET
END_PROPERTY

PROPERTY PUBLIC P_sTwinCAT_Version : STRING
GET
END_GET
END_PROPERTY

END_INTERFACE

// POUs/SYSTEM/FBs/System/FB_SystemDK
//------------------------------------------------------------------------------------------
//                                                                                        	
//***************************** Beckhoff TwinCAT Examples **********************************
//                                                                                        	
//************************************* WARNING ********************************************
// This program is only an example. If it is used as a control program in any real        	
// application, Beckhoff is not responsible for any malfunction, loss or damage           	
// which could arise by using this program!                                               	
//                                                                                        	
//*************************************  Program Info. *************************************
//                                                                                        	
// PLC program name:       	FB_SystemDK (FB)               	                           	
// Hardware platform:      	TwinCat v3.1.4022				                          	
// Modified by:            	Hans Chr. Pallesen 			                                  	
// Email:					h.pallesen@beckhoff.com	                                  	
//                                                                                        	
// ======================================================================================== 
//         Version       Date                        Remarks                              	
// ======================================================================================== 
//         1.0           14 okt 2014                 First release of this example        	
// ======================================================================================== 
//                                                                                        	
//******************************* Aims OF this PLC PROGRAM *********************************
//                                                                                        	
//	TwinCAT device info																	                      	
//                                                                                        	
//----------------------------------------------------------------------------------------- 
FUNCTION_BLOCK FB_SystemDK EXTENDS FB_Basic IMPLEMENTS I_SystemDK
VAR
{attribute 'hide'}
	pInternPointer: POINTER TO INT;
END_VAR
VAR
//**************************
// Property variables
//**************************
	_bIs_ARM: BOOL;
	_stDeviceIdentificationEx: Tc2_Utilities.ST_DeviceIdentificationEx;
	_sTwinCAT_Version: STRING(20);
	_sHardwareSerialNumber: STRING(20);
	
//**********************************
// Methods variable
//**********************************
	FB_SystemDK_M_nEnable_iState: INT;
	FB_SystemDK_M_nEnable_bDone: BOOL; 
	FB_SystemDK_M_nEnable_arrUINT: ARRAY[1..4] OF UINT;
	FB_SystemDK_M_nEnable_stDeviceIdentificationEx: Tc2_Utilities.ST_DeviceIdentificationEx;
	FB_SystemDK_M_nEnable_fb_GetDeviceIdentificationEx: Tc2_Utilities.FB_GetDeviceIdentificationEx;
	FB_SystemDK_M_nEnable_fbADSREAD: Tc2_System.ADSREAD;
	
	FB_SystemDK_M_nCerHost_iState: INT;
	FB_SystemDK_M_nCerHost_sValue: STRING;
	FB_SystemDK_M_nCerHost_fbEnable_R_TRIG: Tc2_Standard.R_TRIG;
	FB_SystemDK_M_nCerHost_fbDisable_R_TRIG: Tc2_Standard.R_TRIG;
	FB_SystemDK_M_nCerHost_fbRegSetValue: Tc2_Utilities.FB_RegSetValue;
	FB_SystemDK_M_nCerHost_fbNT_Reboot: Tc2_Utilities.NT_Reboot;
END_VAR

//	The result of the method is an unsigned double integer
//	0 = idle 
//	1 = coupled
//	2 = starting
//	3 = running
//	4 = aborted
// 	5 = no hardware connected
//  6 = Spare
//	7 = pointer or index error
//	8 = mapping error
//	9 = parameter error
//	10 = complete
//	Any other number = ErrorID
METHOD PUBLIC M_nCerHost : UDINT
VAR_INPUT
	bEnable: BOOL;
	bDisable: BOOL;
END_VAR
//**********************************
// Reset
//**********************************
IF _bReset THEN
	IF _bError THEN
		FB_SystemDK_M_nCerHost_fbRegSetValue(bExecute:= FALSE);
		FB_SystemDK_M_nCerHost_fbNT_Reboot(START:= FALSE); 
		FB_SystemDK_M_nCerHost_iState:= 000;
	END_IF
	M_nReset(bExecute:= _bReset);
END_IF

//**********************************
// Wait for execute
//**********************************
FB_SystemDK_M_nCerHost_fbEnable_R_TRIG(CLK:= bEnable);
IF FB_SystemDK_M_nCerHost_fbEnable_R_TRIG.Q THEN
	FB_SystemDK_M_nCerHost_fbRegSetValue(bExecute:= FALSE);
	FB_SystemDK_M_nCerHost_fbNT_Reboot(START:= FALSE); 
	FB_SystemDK_M_nCerHost_iState:= 001;
END_IF
FB_SystemDK_M_nCerHost_fbDisable_R_TRIG(CLK:= bDisable);
IF FB_SystemDK_M_nCerHost_fbDisable_R_TRIG.Q THEN
	FB_SystemDK_M_nCerHost_fbRegSetValue(bExecute:= FALSE);
	FB_SystemDK_M_nCerHost_fbNT_Reboot(START:= FALSE); 
	FB_SystemDK_M_nCerHost_iState:= 010;
END_IF


//**********************************
// State maschine
//**********************************
CASE FB_SystemDK_M_nCerHost_iState OF
	
	000:	// Do nothing
	
	001:	// Enable CerHost
			M_nCerHost:= cRUNNING;
			FB_SystemDK_M_nCerHost_sValue:= 'CeRDisp.exe';
			FB_SystemDK_M_nCerHost_fbRegSetValue(
				sNetId:= '', 
				sSubKey:= 'init', 
				sValName:= 'Launch90', 
				eValType:= REG_SZ, 
				cbData:= INT_TO_UDINT(Tc2_Standard.LEN(FB_SystemDK_M_nCerHost_sValue)), 
				pData:= ADR(FB_SystemDK_M_nCerHost_sValue), 
				bExecute:= TRUE, 
				tTimeOut:= Tc2_System.DEFAULT_ADS_TIMEOUT, 
				bBusy=> , 
				bError=> , 
				nErrId=> , 
				cbWrite=> );
		
			// Error	
			IF FB_SystemDK_M_nCerHost_fbRegSetValue.bError THEN
				M_nError(nErrorID:= FB_SystemDK_M_nCerHost_fbRegSetValue.nErrId);
				M_nCerHost:= FB_SystemDK_M_nCerHost_fbRegSetValue.nErrId;
			ELSE
				// Done
				IF NOT FB_SystemDK_M_nCerHost_fbRegSetValue.bBusy THEN
					FB_SystemDK_M_nCerHost_fbRegSetValue(bExecute:= FALSE);
					FB_SystemDK_M_nCerHost_iState:= FB_SystemDK_M_nCerHost_iState +1;
				END_IF
			END_IF
	
	002:	// Enable done
			M_nCerHost:= cRUNNING;
			FB_SystemDK_M_nCerHost_iState:= 20;

	010:	// Disable CerHost
			M_nCerHost:= cRUNNING;
			FB_SystemDK_M_nCerHost_sValue:= '_CeRDisp.exe';
			FB_SystemDK_M_nCerHost_fbRegSetValue(
				sNetId:= '', 
				sSubKey:= 'init', 
				sValName:= 'Launch90', 
				eValType:= REG_SZ, 
				cbData:= INT_TO_UDINT(Tc2_Standard.LEN(FB_SystemDK_M_nCerHost_sValue)), 
				pData:= ADR(FB_SystemDK_M_nCerHost_sValue), 
				bExecute:= TRUE, 
				tTimeOut:= Tc2_System.DEFAULT_ADS_TIMEOUT, 
				bBusy=> , 
				bError=> , 
				nErrId=> , 
				cbWrite=> );
		
			// Error	
			IF FB_SystemDK_M_nCerHost_fbRegSetValue.bError THEN
				M_nError(nErrorID:= FB_SystemDK_M_nCerHost_fbRegSetValue.nErrId);
				M_nCerHost:= FB_SystemDK_M_nCerHost_fbRegSetValue.nErrId;
			ELSE
				// Done
				IF NOT FB_SystemDK_M_nCerHost_fbRegSetValue.bBusy THEN
					FB_SystemDK_M_nCerHost_fbRegSetValue(bExecute:= FALSE);
					FB_SystemDK_M_nCerHost_iState:= FB_SystemDK_M_nCerHost_iState +1;
				END_IF
			END_IF
			
	011:	// Disable done
			M_nCerHost:= cRUNNING;
			FB_SystemDK_M_nCerHost_iState:= 20;

	020:	// Reboot
			M_nCerHost:= cRUNNING;
			FB_SystemDK_M_nCerHost_fbNT_Reboot(
				NETID:= '', 
				DELAY:= 0, 
				START:= TRUE, 
				TMOUT:= Tc2_System.DEFAULT_ADS_TIMEOUT, 
				BUSY=> , 
				ERR=> , 
				ERRID=> );
	
			// Error	
			IF FB_SystemDK_M_nCerHost_fbNT_Reboot.ERR THEN
				M_nError(nErrorID:= FB_SystemDK_M_nCerHost_fbNT_Reboot.ERRID);
				M_nCerHost:= FB_SystemDK_M_nCerHost_fbNT_Reboot.ERRID;
			END_IF
		
ELSE
	FB_SystemDK_M_nCerHost_iState:= 000;
END_CASE
END_METHOD

//	The result of the method is an unsigned double integer
//	0 = idle 
//	1 = coupled
//	2 = starting
//	3 = running
//	4 = aborted
// 	5 = no hardware connected
//  6 = Spare
//	7 = pointer or index error
//	8 = mapping error
//	9 = parameter error
//	10 = complete
//	Any other number = ErrorID
METHOD PUBLIC M_nEnable : UDINT
VAR_INPUT
END_VAR
//**********************************
// Reset
//**********************************
IF _bReset THEN
	IF NOT FB_SystemDK_M_nEnable_bDone THEN
		FB_SystemDK_M_nEnable_fb_GetDeviceIdentificationEx(bExecute:= FALSE); 
		FB_SystemDK_M_nEnable_iState:= 000;
	END_IF
	M_nReset(bExecute:= _bReset);
END_IF

// Status
IF _stDeviceIdentificationEx.strHardwareCPU = 'ARM' THEN
	_bIs_ARM:= TRUE;
ELSE
	_bIs_ARM:= FALSE;
END_IF

//**********************************
// State maschine
//**********************************
CASE FB_SystemDK_M_nEnable_iState OF
	
	000:	// Init
			M_nEnable:= cSTARTING;
			FB_SystemDK_M_nEnable_fb_GetDeviceIdentificationEx(bExecute:= FALSE); 
			FB_SystemDK_M_nEnable_fbADSREAD(READ:= FALSE); 
			FB_SystemDK_M_nEnable_bDone:= FALSE;
			FB_SystemDK_M_nEnable_iState:= FB_SystemDK_M_nEnable_iState +1;
		
	001:	// Get data	
			M_nEnable:= cRUNNING;
			FB_SystemDK_M_nEnable_fb_GetDeviceIdentificationEx(bExecute:= FALSE); 
			FB_SystemDK_M_nEnable_fb_GetDeviceIdentificationEx(
				bExecute:= TRUE, 
				tTimeout:= Tc2_System.DEFAULT_ADS_TIMEOUT, 
				sNetId:= '', 
				bBusy=> , 
				bError=> , 
				nErrorID=> , 
				stDevIdent=> FB_SystemDK_M_nEnable_stDeviceIdentificationEx);
	
			FB_SystemDK_M_nEnable_iState:= FB_SystemDK_M_nEnable_iState +1;
	
	002:	// Get data done
			M_nEnable:= cRUNNING;
			FB_SystemDK_M_nEnable_fb_GetDeviceIdentificationEx(bExecute:= TRUE, stDevIdent=> FB_SystemDK_M_nEnable_stDeviceIdentificationEx);
			IF FB_SystemDK_M_nEnable_fb_GetDeviceIdentificationEx.bError THEN
				M_nError(nErrorID:= FB_SystemDK_M_nEnable_fb_GetDeviceIdentificationEx.nErrorID);
				M_nEnable:= FB_SystemDK_M_nEnable_fb_GetDeviceIdentificationEx.nErrorID;
			ELSE
				// Done
				IF NOT FB_SystemDK_M_nEnable_fb_GetDeviceIdentificationEx.bBusy THEN
					_stDeviceIdentificationEx:= FB_SystemDK_M_nEnable_stDeviceIdentificationEx;
					FB_SystemDK_M_nEnable_fb_GetDeviceIdentificationEx(bExecute:= FALSE); 
					FB_SystemDK_M_nEnable_iState:= FB_SystemDK_M_nEnable_iState +1;
				END_IF	
			END_IF
		
	003:	// Read 
			M_nEnable:= cRUNNING;
			FB_SystemDK_M_nEnable_fbADSREAD(
				NETID:= , 
				PORT:= 10000, 
				IDXGRP:= 160, 
				IDXOFFS:= 0, 
				LEN:= SIZEOF(FB_SystemDK_M_nEnable_arrUINT), 
				DESTADDR:= ADR(FB_SystemDK_M_nEnable_arrUINT), 
				READ:= TRUE, 
				TMOUT:= , 
				BUSY=> , 
				ERR=> , 
				ERRID=> );
						
			IF NOT FB_SystemDK_M_nEnable_fbADSREAD.BUSY THEN
				_sTwinCAT_Version:= 'v';
				_sTwinCAT_Version:= Tc2_Standard.CONCAT(_sTwinCAT_Version, UINT_TO_STRING(FB_SystemDK_M_nEnable_arrUINT[2]));
				_sTwinCAT_Version:= Tc2_Standard.CONCAT(_sTwinCAT_Version, '.');
				_sTwinCAT_Version:= Tc2_Standard.CONCAT(_sTwinCAT_Version, UINT_TO_STRING(FB_SystemDK_M_nEnable_arrUINT[1]));
				_sTwinCAT_Version:= Tc2_Standard.CONCAT(_sTwinCAT_Version, '.');
				_sTwinCAT_Version:= Tc2_Standard.CONCAT(_sTwinCAT_Version, UINT_TO_STRING(FB_SystemDK_M_nEnable_arrUINT[4]));
				_sTwinCAT_Version:= Tc2_Standard.CONCAT(_sTwinCAT_Version, '.');
				_sTwinCAT_Version:= Tc2_Standard.CONCAT(_sTwinCAT_Version, UINT_TO_STRING(FB_SystemDK_M_nEnable_arrUINT[3]));
				FB_SystemDK_M_nEnable_iState:= FB_SystemDK_M_nEnable_iState +1;
			END_IF

	004:	// Device HardwareSerialNumber	
			M_nEnable:= cRUNNING;
			_sHardwareSerialNumber:= _stDeviceIdentificationEx.strHardwareSerialNo;
			FB_SystemDK_M_nEnable_iState:= FB_SystemDK_M_nEnable_iState +1;
			
	005:	// Done	
			M_nEnable:= cCOMPLETE;
			FB_SystemDK_M_nEnable_bDone:= TRUE;

ELSE
	FB_SystemDK_M_nEnable_iState:= 000;
END_CASE


// bReady
IF FB_SystemDK_M_nEnable_bDone THEN
	_bReady:= TRUE;
ELSE
	_bReady:= FALSE;
END_IF
END_METHOD

METHOD PUBLIC M_nGetTimeStampInMs : ULINT
VAR_INPUT
END_VAR
M_nGetTimeStampInMs:= Tc2_EtherCAT.F_GetCurDcTaskTime64() / EC_DCTIME_TICKSPERMSEC64;
END_METHOD

{attribute 'monitoring' := 'variable'}
PROPERTY PUBLIC P_bIs_ARM : BOOL
GET
P_bIs_ARM:= _bIs_ARM;
END_GET
END_PROPERTY

{attribute 'monitoring' := 'variable'}
PROPERTY PUBLIC P_bIs_CE_Device : BOOL
GET
P_bIs_CE_Device:= _stDeviceIdentificationEx.strImageOsName = 'Windows CE';
END_GET
END_PROPERTY

{attribute 'monitoring' := 'variable'}
PROPERTY PUBLIC P_bIs_x64 : BOOL
GET
IF _bIs_ARM THEN
	P_bIs_x64:= FALSE;
ELSE
	IF SIZEOF(pInternPointer) > 4 THEN
		P_bIs_x64:= TRUE;
	ELSE
		P_bIs_x64:= FALSE;
	END_IF	
END_IF
END_GET
END_PROPERTY

{attribute 'monitoring' := 'variable'}
PROPERTY PUBLIC P_bIs_x86 : BOOL
GET
IF _bIs_ARM THEN
	P_bIs_x86:= FALSE;
ELSE
	IF SIZEOF(pInternPointer) = 4 THEN
		P_bIs_x86:= TRUE;
	ELSE
		P_bIs_x86:= FALSE;
	END_IF	
END_IF
END_GET
END_PROPERTY

{attribute 'monitoring' := 'variable'}
PROPERTY PUBLIC P_nAdsPort : UINT
GET
P_nAdsPort:= TwinCAT_SystemInfoVarList._AppInfo.AdsPort;
END_GET
END_PROPERTY

{attribute 'monitoring' := 'variable'}
PROPERTY PUBLIC P_nCycleTime : UDINT
GET
P_nCycleTime:= TwinCAT_SystemInfoVarList._TaskInfo[Tc2_System.GETCURTASKINDEXEX()].CycleTime;
END_GET
END_PROPERTY

{attribute 'monitoring' := 'variable'}
PROPERTY PUBLIC P_sHardwareSerialNumber : String
GET
P_sHardwareSerialNumber:= _sHardwareSerialNumber;
END_GET
END_PROPERTY

{attribute 'monitoring' := 'variable'}
PROPERTY PUBLIC P_stDeviceIdentificationEx : Tc2_Utilities.ST_DeviceIdentificationEx
GET
P_stDeviceIdentificationEx:= _stDeviceIdentificationEx;
END_GET
END_PROPERTY

{attribute 'monitoring' := 'variable'}
PROPERTY PUBLIC P_sTwinCAT_Version : STRING
GET
P_sTwinCAT_Version:= _sTwinCAT_Version;
END_GET
END_PROPERTY

END_FUNCTION_BLOCK
